LIN {X 0,Y 474.661,Z 275.668,A -85,B 0,C 180,E1 -7353.629,E2 -7353.629} C_VEL
LIN {X 0,Y 474.637,Z 275.665,A -85,B 0,C 180,E1 -7356.642,E2 -7356.642} C_VEL
LIN {X 0,Y 474.656,Z 275.67,A -85,B 0,C 180,E1 -7360.09,E2 -7360.09} C_VEL
LIN {X 0,Y 474.648,Z 275.66,A -85,B 0,C 180,E1 -7362.775,E2 -7362.775} C_VEL
LIN {X 0,Y 474.647,Z 275.67,A -85,B 0,C 180,E1 -7365.421,E2 -7365.421} C_VEL
LIN {X 0,Y 474.706,Z 275.661,A -85,B 0,C 180,E1 -7368.038,E2 -7368.038} C_VEL
LIN {X 0,Y 474.71,Z 275.661,A -85,B 0,C 180,E1 -7371.487,E2 -7371.487} C_VEL
LIN {X 0,Y 474.743,Z 275.645,A -85,B 0,C 180,E1 -7374.905,E2 -7374.905} C_VEL
LIN {X 0,Y 474.887,Z 275.637,A -85,B 0,C 180,E1 -7377.456,E2 -7377.456} C_VEL
LIN {X 0,Y 474.911,Z 275.639,A -85,B 0,C 180,E1 -7380,E2 -7380} C_VEL
LIN {X 0,Y 474.877,Z 275.632,A -85,B 0,C 180,E1 -7382.545,E2 -7382.545} C_VEL
LIN {X 0,Y 474.749,Z 275.66,A -85,B 0,C 180,E1 -7385.948,E2 -7385.948} C_VEL
LIN {X 0,Y 474.698,Z 275.655,A -85,B 0,C 180,E1 -7388.515,E2 -7388.515} C_VEL
LIN {X 0,Y 474.707,Z 275.667,A -85,B 0,C 180,E1 -7391.963,E2 -7391.963} C_VEL
LIN {X 0,Y 474.691,Z 275.662,A -85,B 0,C 180,E1 -7395.456,E2 -7395.456} C_VEL
LIN {X 0,Y 474.661,Z 275.656,A -85,B 0,C 180,E1 -7399.011,E2 -7399.011} C_VEL
LIN {X 0,Y 474.586,Z 275.681,A -85,B 0,C 180,E1 -7401.73,E2 -7401.73} C_VEL
LIN {X 0,Y 474.623,Z 275.67,A -85,B 0,C 180,E1 -7404.495,E2 -7404.495} C_VEL
LIN {X 0,Y 474.595,Z 275.676,A -85,B 0,C 180,E1 -7407.327,E2 -7407.327} C_VEL
LIN {X 0,Y 474.553,Z 275.688,A -85,B 0,C 180,E1 -7410.234,E2 -7410.234} C_VEL
LIN {X 0,Y 474.61,Z 275.676,A -85,B 0,C 180,E1 -7413.223,E2 -7413.223} C_VEL
LIN {X 0,Y 474.565,Z 275.685,A -85,B 0,C 180,E1 -7416.326,E2 -7416.326} C_VEL
LIN {X 0,Y 474.6,Z 275.68,A -85,B 0,C 180,E1 -7419.551,E2 -7419.551} C_VEL
LIN {X 0,Y 474.568,Z 275.682,A -85,B 0,C 180,E1 -7422.94,E2 -7422.94} C_VEL
LIN {X 0,Y 474.582,Z 275.68,A -85,B 0,C 180,E1 -7425.892,E2 -7425.892} C_VEL
LIN {X 0,Y 474.598,Z 275.757,A -85,B 0,C 180,E1 -7426.52,E2 -7426.52} C_VEL
LIN {X 0,Y 477.677,Z 285.882,A -85,B 0,C 180,E1 -7428.043,E2 -7428.043} C_VEL
LIN {X 0,Y 486.034,Z 303.231,A -85,B 0,C 180,E1 -7428.924,E2 -7428.924} C_VEL
LIN {X 0,Y 486.81,Z 305.51,A -85,B 0,C 180,E1 -7429.015,E2 -7429.015} C_VEL
LIN {X 0,Y 484.879,Z 443.516,A -85,B 0,C 180,E1 -7431.179,E2 -7431.179} C_VEL
LIN {X 0,Y 484.222,Z 449.369,A -85,B 0,C 180,E1 -7431.235,E2 -7431.235} C_VEL
LIN {X 0,Y 478.792,Z 468.46,A -85,B 0,C 180,E1 -7431.216,E2 -7431.216} C_VEL
LIN {X 0,Y 478.144,Z 474.313,A -85,B 0,C 180,E1 -7431.273,E2 -7431.273} C_VEL
LIN {X 0,Y 477.665,Z 496.241,A -85,B 0,C 180,E1 -7431.674,E2 -7431.674} C_VEL
LIN {X 0,Y 477.021,Z 512.96,A -85,B 0,C 180,E1 -7432.157,E2 -7432.157} C_VEL
LIN {X 0,Y 476.29,Z 528.431,A -85,B 0,C 180,E1 -7432.772,E2 -7432.772} C_VEL
LIN {X 0,Y 475.249,Z 544.663,A -85,B 0,C 180,E1 -7433.609,E2 -7433.609} C_VEL
LIN {X 0,Y 474.176,Z 559.577,A -85,B 0,C 180,E1 -7434.57,E2 -7434.57} C_VEL
LIN {X 0,Y 473.106,Z 573.275,A -85,B 0,C 180,E1 -7435.633,E2 -7435.633} C_VEL
LIN {X 0,Y 472.039,Z 586.323,A -85,B 0,C 180,E1 -7436.828,E2 -7436.828} C_VEL
LIN {X 0,Y 470.902,Z 599.014,A -85,B 0,C 180,E1 -7438.202,E2 -7438.202} C_VEL
LIN {X 0,Y 469.898,Z 610.493,A -85,B 0,C 180,E1 -7439.669,E2 -7439.669} C_VEL
LIN {X 0,Y 468.991,Z 621.639,A -85,B 0,C 180,E1 -7441.345,E2 -7441.345} C_VEL
LIN {X 0,Y 468.276,Z 630.97,A -85,B 0,C 180,E1 -7442.999,E2 -7442.999} C_VEL
LIN {X 0,Y 467.695,Z 639.197,A -85,B 0,C 180,E1 -7444.723,E2 -7444.723} C_VEL
LIN {X 0,Y 467.236,Z 646.457,A -85,B 0,C 180,E1 -7446.57,E2 -7446.57} C_VEL
LIN {X 0,Y 466.954,Z 652.215,A -85,B 0,C 180,E1 -7448.362,E2 -7448.362} C_VEL
LIN {X 0,Y 466.777,Z 656.937,A -85,B 0,C 180,E1 -7450.198,E2 -7450.198} C_VEL
LIN {X 0,Y 466.576,Z 661.108,A -85,B 0,C 180,E1 -7452.467,E2 -7452.467} C_VEL
LIN {X 0,Y 466.537,Z 663.472,A -85,B 0,C 180,E1 -7454.605,E2 -7454.605} C_VEL
LIN {X 0,Y 466.502,Z 664.25,A -85,B 0,C 180,E1 -7456.052,E2 -7456.052} C_VEL
LIN {X 0,Y 466.647,Z 664.195,A -85,B 0,C 180,E1 -7458.224,E2 -7458.224} C_VEL
LIN {X 0,Y 466.535,Z 662.564,A -85,B 0,C 180,E1 -7460.462,E2 -7460.462} C_VEL
LIN {X 0,Y 466.638,Z 660.118,A -85,B 0,C 180,E1 -7462.21,E2 -7462.21} C_VEL
LIN {X 0,Y 466.834,Z 656.756,A -85,B 0,C 180,E1 -7463.951,E2 -7463.951} C_VEL
LIN {X 0,Y 467.026,Z 651.048,A -85,B 0,C 180,E1 -7466.117,E2 -7466.117} C_VEL
LIN {X 0,Y 467.344,Z 643.603,A -85,B 0,C 180,E1 -7468.276,E2 -7468.276} C_VEL
LIN {X 0,Y 467.92,Z 635.211,A -85,B 0,C 180,E1 -7470.215,E2 -7470.215} C_VEL
LIN {X 0,Y 468.5,Z 626.235,A -85,B 0,C 180,E1 -7471.934,E2 -7471.934} C_VEL
LIN {X 0,Y 469.405,Z 615.604,A -85,B 0,C 180,E1 -7473.648,E2 -7473.648} C_VEL
LIN {X 0,Y 470.337,Z 604.684,A -85,B 0,C 180,E1 -7475.144,E2 -7475.144} C_VEL
LIN {X 0,Y 471.253,Z 593.821,A -85,B 0,C 180,E1 -7476.422,E2 -7476.422} C_VEL
LIN {X 0,Y 472.226,Z 581.157,A -85,B 0,C 180,E1 -7477.697,E2 -7477.697} C_VEL
LIN {X 0,Y 473.302,Z 567.479,A -85,B 0,C 180,E1 -7478.862,E2 -7478.862} C_VEL
LIN {X 0,Y 474.306,Z 554.277,A -85,B 0,C 180,E1 -7479.811,E2 -7479.811} C_VEL
LIN {X 0,Y 475.239,Z 540.053,A -85,B 0,C 180,E1 -7480.653,E2 -7480.653} C_VEL
LIN {X 0,Y 476.07,Z 524.768,A -85,B 0,C 180,E1 -7481.388,E2 -7481.388} C_VEL
LIN {X 0,Y 476.866,Z 508.398,A -85,B 0,C 180,E1 -7481.988,E2 -7481.988} C_VEL
LIN {X 0,Y 477.425,Z 492.53,A -85,B 0,C 180,E1 -7482.405,E2 -7482.405} C_VEL
LIN {X 0,Y 478.233,Z 435.094,A -85,B 0,C 180,E1 -7483.329,E2 -7483.329} C_VEL
LIN {X 0,Y 480.033,Z 307.307,A -85,B 0,C 180,E1 -7485.325,E2 -7485.325} C_VEL
LIN {X 0,Y 473.3,Z 292.179,A -85,B 0,C 180,E1 -7485.994,E2 -7485.994} C_VEL
LIN {X 0,Y 470.234,Z 285.606,A -85,B 0,C 180,E1 -7486.308,E2 -7486.308} C_VEL
LIN {X 0,Y 467.603,Z 276.551,A -85,B 0,C 180,E1 -7487.634,E2 -7487.634} C_VEL
LIN {X 0,Y 467.623,Z 276.551,A -85,B 0,C 180,E1 -7490.223,E2 -7490.223} C_VEL
LIN {X 0,Y 467.558,Z 276.562,A -85,B 0,C 180,E1 -7493.944,E2 -7493.944} C_VEL
LIN {X 0,Y 467.529,Z 276.559,A -85,B 0,C 180,E1 -7496.806,E2 -7496.806} C_VEL
LIN {X 0,Y 467.538,Z 276.559,A -85,B 0,C 180,E1 -7499.739,E2 -7499.739} C_VEL
LIN {X 0,Y 467.552,Z 276.556,A -85,B 0,C 180,E1 -7502.761,E2 -7502.761} C_VEL
LIN {X 0,Y 467.538,Z 276.558,A -85,B 0,C 180,E1 -7505.891,E2 -7505.891} C_VEL
LIN {X 0,Y 467.527,Z 276.555,A -85,B 0,C 180,E1 -7509.15,E2 -7509.15} C_VEL
LIN {X 0,Y 467.551,Z 276.554,A -85,B 0,C 180,E1 -7511.406,E2 -7511.406} C_VEL
LIN {X 0,Y 467.564,Z 276.552,A -85,B 0,C 180,E1 -7515.051,E2 -7515.051} C_VEL
LIN {X 0,Y 467.551,Z 276.554,A -85,B 0,C 180,E1 -7518.727,E2 -7518.727} C_VEL
LIN {X 0,Y 467.54,Z 276.54,A -85,B 0,C 180,E1 -7521.952,E2 -7521.952} C_VEL
LIN {X 0,Y 467.551,Z 276.54,A -85,B 0,C 180,E1 -7525.166,E2 -7525.166} C_VEL
LIN {X 0,Y 467.559,Z 276.555,A -85,B 0,C 180,E1 -7528.257,E2 -7528.257} C_VEL
LIN {X 0,Y 467.544,Z 276.548,A -85,B 0,C 180,E1 -7531.248,E2 -7531.248} C_VEL
LIN {X 0,Y 467.577,Z 276.549,A -85,B 0,C 180,E1 -7534.401,E2 -7534.401} C_VEL
LIN {X 0,Y 467.577,Z 276.544,A -85,B 0,C 180,E1 -7536.995,E2 -7536.995} C_VEL
LIN {X 0,Y 467.623,Z 276.549,A -85,B 0,C 180,E1 -7539.777,E2 -7539.777} C_VEL
LIN {X 0,Y 467.595,Z 276.541,A -85,B 0,C 180,E1 -7542.506,E2 -7542.506} C_VEL
LIN {X 0,Y 467.602,Z 276.55,A -85,B 0,C 180,E1 -7545.196,E2 -7545.196} C_VEL
LIN {X 0,Y 467.658,Z 276.536,A -85,B 0,C 180,E1 -7547.854,E2 -7547.854} C_VEL
LIN {X 0,Y 467.669,Z 276.544,A -85,B 0,C 180,E1 -7551.357,E2 -7551.357} C_VEL
LIN {X 0,Y 467.736,Z 276.524,A -85,B 0,C 180,E1 -7553.962,E2 -7553.962} C_VEL
LIN {X 0,Y 467.849,Z 276.524,A -85,B 0,C 180,E1 -7557.417,E2 -7557.417} C_VEL
LIN {X 0,Y 467.882,Z 276.504,A -85,B 0,C 180,E1 -7560,E2 -7560} C_VEL
LIN {X 0,Y 467.859,Z 276.514,A -85,B 0,C 180,E1 -7562.582,E2 -7562.582} C_VEL
LIN {X 0,Y 467.724,Z 276.523,A -85,B 0,C 180,E1 -7566.037,E2 -7566.037} C_VEL
LIN {X 0,Y 467.682,Z 276.532,A -85,B 0,C 180,E1 -7568.642,E2 -7568.642} C_VEL
LIN {X 0,Y 467.656,Z 276.538,A -85,B 0,C 180,E1 -7572.145,E2 -7572.145} C_VEL
LIN {X 0,Y 467.639,Z 276.544,A -85,B 0,C 180,E1 -7575.695,E2 -7575.695} C_VEL
LIN {X 0,Y 467.622,Z 276.55,A -85,B 0,C 180,E1 -7579.307,E2 -7579.307} C_VEL
LIN {X 0,Y 467.534,Z 276.555,A -85,B 0,C 180,E1 -7582.073,E2 -7582.073} C_VEL
LIN {X 0,Y 467.604,Z 276.554,A -85,B 0,C 180,E1 -7584.887,E2 -7584.887} C_VEL
LIN {X 0,Y 467.619,Z 276.544,A -85,B 0,C 180,E1 -7587.769,E2 -7587.769} C_VEL
LIN {X 0,Y 467.567,Z 276.557,A -85,B 0,C 180,E1 -7591.045,E2 -7591.045} C_VEL
LIN {X 0,Y 467.588,Z 276.55,A -85,B 0,C 180,E1 -7594.242,E2 -7594.242} C_VEL
LIN {X 0,Y 467.549,Z 276.554,A -85,B 0,C 180,E1 -7597.186,E2 -7597.186} C_VEL
LIN {X 0,Y 467.577,Z 276.55,A -85,B 0,C 180,E1 -7600.264,E2 -7600.264} C_VEL
LIN {X 0,Y 467.585,Z 276.554,A -85,B 0,C 180,E1 -7602.567,E2 -7602.567} C_VEL
LIN {X 0,Y 467.569,Z 276.555,A -85,B 0,C 180,E1 -7605.053,E2 -7605.053} C_VEL
LIN {X 0,Y 467.587,Z 276.549,A -85,B 0,C 180,E1 -7607.44,E2 -7607.44} C_VEL
LIN {X 0,Y 467.581,Z 276.556,A -85,B 0,C 180,E1 -7610.855,E2 -7610.855} C_VEL
LIN {X 0,Y 467.558,Z 276.554,A -85,B 0,C 180,E1 -7614.261,E2 -7614.261} C_VEL
LIN {X 0,Y 467.62,Z 276.653,A -85,B 0,C 180,E1 -7616.939,E2 -7616.939} C_VEL
LIN {X 0,Y 474.089,Z 297.974,A -85,B 0,C 180,E1 -7619.734,E2 -7619.734} C_VEL
LIN {X 0,Y 475.758,Z 304.134,A -85,B 0,C 180,E1 -7620.503,E2 -7620.503} C_VEL
LIN {X 0,Y 475.416,Z 309.361,A -85,B 0,C 180,E1 -7621.045,E2 -7621.045} C_VEL
LIN {X 0,Y 479.849,Z 335.021,A -85,B 0,C 180,E1 -7621.748,E2 -7621.748} C_VEL
LIN {X 0,Y 477.322,Z 515.075,A -85,B 0,C 180,E1 -7624.569,E2 -7624.569} C_VEL
LIN {X 0,Y 476.755,Z 530.976,A -85,B 0,C 180,E1 -7624.954,E2 -7624.954} C_VEL
LIN {X 0,Y 476.072,Z 547.463,A -85,B 0,C 180,E1 -7625.527,E2 -7625.527} C_VEL
LIN {X 0,Y 475.182,Z 561.942,A -85,B 0,C 180,E1 -7626.174,E2 -7626.174} C_VEL
LIN {X 0,Y 474.26,Z 575.705,A -85,B 0,C 180,E1 -7626.948,E2 -7626.948} C_VEL
LIN {X 0,Y 473.097,Z 590.803,A -85,B 0,C 180,E1 -7627.97,E2 -7627.97} C_VEL
LIN {X 0,Y 472.056,Z 604.285,A -85,B 0,C 180,E1 -7629.065,E2 -7629.065} C_VEL
LIN {X 0,Y 470.947,Z 618.3,A -85,B 0,C 180,E1 -7630.426,E2 -7630.426} C_VEL
LIN {X 0,Y 470.025,Z 629.422,A -85,B 0,C 180,E1 -7631.7,E2 -7631.7} C_VEL
LIN {X 0,Y 469.126,Z 640.999,A -85,B 0,C 180,E1 -7633.239,E2 -7633.239} C_VEL
LIN {X 0,Y 468.442,Z 650.925,A -85,B 0,C 180,E1 -7634.779,E2 -7634.779} C_VEL
LIN {X 0,Y 467.748,Z 660.458,A -85,B 0,C 180,E1 -7636.533,E2 -7636.533} C_VEL
LIN {X 0,Y 467.359,Z 668.439,A -85,B 0,C 180,E1 -7638.287,E2 -7638.287} C_VEL
LIN {X 0,Y 466.981,Z 675.094,A -85,B 0,C 180,E1 -7640.034,E2 -7640.034} C_VEL
LIN {X 0,Y 466.833,Z 680.492,A -85,B 0,C 180,E1 -7641.778,E2 -7641.778} C_VEL
LIN {X 0,Y 466.748,Z 684.944,A -85,B 0,C 180,E1 -7643.607,E2 -7643.607} C_VEL
LIN {X 0,Y 466.605,Z 688.611,A -85,B 0,C 180,E1 -7645.681,E2 -7645.681} C_VEL
LIN {X 0,Y 466.637,Z 690.554,A -85,B 0,C 180,E1 -7647.41,E2 -7647.41} C_VEL
LIN {X 0,Y 466.614,Z 691.515,A -85,B 0,C 180,E1 -7649.137,E2 -7649.137} C_VEL
LIN {X 0,Y 466.615,Z 691.51,A -85,B 0,C 180,E1 -7650.863,E2 -7650.863} C_VEL
LIN {X 0,Y 466.637,Z 690.539,A -85,B 0,C 180,E1 -7652.59,E2 -7652.59} C_VEL
LIN {X 0,Y 466.606,Z 688.587,A -85,B 0,C 180,E1 -7654.319,E2 -7654.319} C_VEL
LIN {X 0,Y 466.748,Z 684.913,A -85,B 0,C 180,E1 -7656.394,E2 -7656.394} C_VEL
LIN {X 0,Y 466.794,Z 680.451,A -85,B 0,C 180,E1 -7658.223,E2 -7658.223} C_VEL
LIN {X 0,Y 466.981,Z 675.045,A -85,B 0,C 180,E1 -7659.967,E2 -7659.967} C_VEL
LIN {X 0,Y 467.359,Z 668.384,A -85,B 0,C 180,E1 -7661.713,E2 -7661.713} C_VEL
LIN {X 0,Y 467.741,Z 660.409,A -85,B 0,C 180,E1 -7663.468,E2 -7663.468} C_VEL
LIN {X 0,Y 468.436,Z 650.897,A -85,B 0,C 180,E1 -7665.222,E2 -7665.222} C_VEL
LIN {X 0,Y 469.265,Z 639.518,A -85,B 0,C 180,E1 -7666.98,E2 -7666.98} C_VEL
LIN {X 0,Y 470.235,Z 627.72,A -85,B 0,C 180,E1 -7668.518,E2 -7668.518} C_VEL
LIN {X 0,Y 471.238,Z 615.457,A -85,B 0,C 180,E1 -7669.884,E2 -7669.884} C_VEL
LIN {X 0,Y 472.335,Z 602.13,A -85,B 0,C 180,E1 -7671.151,E2 -7671.151} C_VEL
LIN {X 0,Y 473.386,Z 588.501,A -85,B 0,C 180,E1 -7672.246,E2 -7672.246} C_VEL
LIN {X 0,Y 474.485,Z 574.417,A -85,B 0,C 180,E1 -7673.183,E2 -7673.183} C_VEL
LIN {X 0,Y 475.561,Z 558.809,A -85,B 0,C 180,E1 -7674.037,E2 -7674.037} C_VEL
LIN {X 0,Y 476.477,Z 543.201,A -85,B 0,C 180,E1 -7674.713,E2 -7674.713} C_VEL
LIN {X 0,Y 477.276,Z 526.491,A -85,B 0,C 180,E1 -7675.25,E2 -7675.25} C_VEL
LIN {X 0,Y 477.79,Z 509.954,A -85,B 0,C 180,E1 -7675.603,E2 -7675.603} C_VEL
LIN {X 0,Y 480.42,Z 335.028,A -85,B 0,C 180,E1 -7678.373,E2 -7678.373} C_VEL
LIN {X 0,Y 476.597,Z 313.02,A -85,B 0,C 180,E1 -7679.018,E2 -7679.018} C_VEL
LIN {X 0,Y 475.858,Z 308.841,A -85,B 0,C 180,E1 -7679.169,E2 -7679.169} C_VEL
LIN {X 0,Y 476.125,Z 304.227,A -85,B 0,C 180,E1 -7679.665,E2 -7679.665} C_VEL
LIN {X 0,Y 471.964,Z 289.925,A -85,B 0,C 180,E1 -7681.599,E2 -7681.599} C_VEL
LIN {X 0,Y 467.609,Z 276.551,A -85,B 0,C 180,E1 -7683.56,E2 -7683.56} C_VEL
LIN {X 0,Y 467.528,Z 276.557,A -85,B 0,C 180,E1 -7686.962,E2 -7686.962} C_VEL
LIN {X 0,Y 467.582,Z 276.553,A -85,B 0,C 180,E1 -7689.955,E2 -7689.955} C_VEL
LIN {X 0,Y 467.586,Z 276.546,A -85,B 0,C 180,E1 -7692.567,E2 -7692.567} C_VEL
LIN {X 0,Y 467.57,Z 276.549,A -85,B 0,C 180,E1 -7695.054,E2 -7695.054} C_VEL
LIN {X 0,Y 467.588,Z 276.549,A -85,B 0,C 180,E1 -7697.44,E2 -7697.44} C_VEL
LIN {X 0,Y 467.582,Z 276.557,A -85,B 0,C 180,E1 -7700.856,E2 -7700.856} C_VEL
LIN {X 0,Y 467.559,Z 276.553,A -85,B 0,C 180,E1 -7704.261,E2 -7704.261} C_VEL
LIN {X 0,Y 467.582,Z 276.545,A -85,B 0,C 180,E1 -7707.321,E2 -7707.321} C_VEL
LIN {X 0,Y 467.57,Z 276.55,A -85,B 0,C 180,E1 -7710.668,E2 -7710.668} C_VEL
LIN {X 0,Y 467.618,Z 276.546,A -85,B 0,C 180,E1 -7713.2,E2 -7713.2} C_VEL
LIN {X 0,Y 467.594,Z 276.544,A -85,B 0,C 180,E1 -7716.469,E2 -7716.469} C_VEL
LIN {X 0,Y 467.624,Z 276.545,A -85,B 0,C 180,E1 -7719.778,E2 -7719.778} C_VEL
LIN {X 0,Y 467.607,Z 276.539,A -85,B 0,C 180,E1 -7722.507,E2 -7722.507} C_VEL
LIN {X 0,Y 467.606,Z 276.549,A -85,B 0,C 180,E1 -7725.197,E2 -7725.197} C_VEL
LIN {X 0,Y 467.658,Z 276.538,A -85,B 0,C 180,E1 -7727.855,E2 -7727.855} C_VEL
LIN {X 0,Y 467.669,Z 276.539,A -85,B 0,C 180,E1 -7731.357,E2 -7731.357} C_VEL
LIN {X 0,Y 467.715,Z 276.533,A -85,B 0,C 180,E1 -7733.963,E2 -7733.963} C_VEL
LIN {X 0,Y 467.852,Z 276.513,A -85,B 0,C 180,E1 -7737.418,E2 -7737.418} C_VEL
LIN {X 0,Y 467.88,Z 276.515,A -85,B 0,C 180,E1 -7740,E2 -7740} C_VEL
LIN {X 0,Y 467.817,Z 276.511,A -85,B 0,C 180,E1 -7742.584,E2 -7742.584} C_VEL
LIN {X 0,Y 467.712,Z 276.538,A -85,B 0,C 180,E1 -7746.038,E2 -7746.038} C_VEL
LIN {X 0,Y 467.659,Z 276.532,A -85,B 0,C 180,E1 -7748.644,E2 -7748.644} C_VEL
LIN {X 0,Y 467.659,Z 276.542,A -85,B 0,C 180,E1 -7752.146,E2 -7752.146} C_VEL
LIN {X 0,Y 467.616,Z 276.545,A -85,B 0,C 180,E1 -7755.696,E2 -7755.696} C_VEL
LIN {X 0,Y 467.621,Z 276.532,A -85,B 0,C 180,E1 -7759.308,E2 -7759.308} C_VEL
LIN {X 0,Y 467.529,Z 276.562,A -85,B 0,C 180,E1 -7762.075,E2 -7762.075} C_VEL
LIN {X 0,Y 467.553,Z 276.552,A -85,B 0,C 180,E1 -7764.891,E2 -7764.891} C_VEL
LIN {X 0,Y 467.54,Z 276.553,A -85,B 0,C 180,E1 -7767.775,E2 -7767.775} C_VEL
LIN {X 0,Y 467.53,Z 276.557,A -85,B 0,C 180,E1 -7771.037,E2 -7771.037} C_VEL
LIN {X 0,Y 467.564,Z 276.557,A -85,B 0,C 180,E1 -7774.237,E2 -7774.237} C_VEL
LIN {X 0,Y 467.511,Z 276.564,A -85,B 0,C 180,E1 -7777.18,E2 -7777.18} C_VEL
LIN {X 0,Y 467.52,Z 276.561,A -85,B 0,C 180,E1 -7780.271,E2 -7780.271} C_VEL
LIN {X 0,Y 467.519,Z 276.561,A -85,B 0,C 180,E1 -7782.569,E2 -7782.569} C_VEL
LIN {X 0,Y 467.557,Z 276.554,A -85,B 0,C 180,E1 -7785.878,E2 -7785.878} C_VEL
LIN {X 0,Y 467.571,Z 276.74,A -85,B 0,C 180,E1 -7786.065,E2 -7786.065} C_VEL
LIN {X 0,Y 470.647,Z 286.352,A -85,B 0,C 180,E1 -7787.53,E2 -7787.53} C_VEL
LIN {X 0,Y 479.664,Z 304.887,A -85,B 0,C 180,E1 -7788.511,E2 -7788.511} C_VEL
LIN {X 0,Y 480.616,Z 306.974,A -85,B 0,C 180,E1 -7788.614,E2 -7788.614} C_VEL
LIN {X 0,Y 479.557,Z 380.616,A -85,B 0,C 180,E1 -7789.793,E2 -7789.793} C_VEL
LIN {X 0,Y 478.144,Z 474.313,A -85,B 0,C 180,E1 -7791.273,E2 -7791.273} C_VEL
LIN {X 0,Y 477.526,Z 480.156,A -85,B 0,C 180,E1 -7791.331,E2 -7791.331} C_VEL
LIN {X 0,Y 472.521,Z 497.266,A -85,B 0,C 180,E1 -7791.378,E2 -7791.378} C_VEL
LIN {X 0,Y 471.265,Z 503.014,A -85,B 0,C 180,E1 -7791.462,E2 -7791.462} C_VEL
LIN {X 0,Y 471.06,Z 504.923,A -85,B 0,C 180,E1 -7791.512,E2 -7791.512} C_VEL
LIN {X 0,Y 470.373,Z 519.803,A -85,B 0,C 180,E1 -7792.019,E2 -7792.019} C_VEL
LIN {X 0,Y 469.458,Z 534.84,A -85,B 0,C 180,E1 -7792.7,E2 -7792.7} C_VEL
LIN {X 0,Y 468.47,Z 549.447,A -85,B 0,C 180,E1 -7793.526,E2 -7793.526} C_VEL
LIN {X 0,Y 467.331,Z 564.147,A -85,B 0,C 180,E1 -7794.539,E2 -7794.539} C_VEL
LIN {X 0,Y 466.144,Z 578.17,A -85,B 0,C 180,E1 -7795.702,E2 -7795.702} C_VEL
LIN {X 0,Y 464.881,Z 591.514,A -85,B 0,C 180,E1 -7797.027,E2 -7797.027} C_VEL
LIN {X 0,Y 463.723,Z 603.844,A -85,B 0,C 180,E1 -7798.475,E2 -7798.475} C_VEL
LIN {X 0,Y 462.667,Z 615.421,A -85,B 0,C 180,E1 -7800.075,E2 -7800.075} C_VEL
LIN {X 0,Y 461.861,Z 624.919,A -85,B 0,C 180,E1 -7801.607,E2 -7801.607} C_VEL
LIN {X 0,Y 461.041,Z 634.892,A -85,B 0,C 180,E1 -7803.52,E2 -7803.52} C_VEL
LIN {X 0,Y 460.508,Z 642.099,A -85,B 0,C 180,E1 -7805.185,E2 -7805.185} C_VEL
LIN {X 0,Y 460.099,Z 648.942,A -85,B 0,C 180,E1 -7807.076,E2 -7807.076} C_VEL
LIN {X 0,Y 459.847,Z 654.016,A -85,B 0,C 180,E1 -7808.795,E2 -7808.795} C_VEL
LIN {X 0,Y 459.669,Z 657.665,A -85,B 0,C 180,E1 -7810.344,E2 -7810.344} C_VEL
LIN {X 0,Y 459.506,Z 660.994,A -85,B 0,C 180,E1 -7812.188,E2 -7812.188} C_VEL
LIN {X 0,Y 459.461,Z 663.629,A -85,B 0,C 180,E1 -7814.508,E2 -7814.508} C_VEL
LIN {X 0,Y 459.422,Z 664.407,A -85,B 0,C 180,E1 -7815.832,E2 -7815.832} C_VEL
LIN {X 0,Y 459.561,Z 664.425,A -85,B 0,C 180,E1 -7818.168,E2 -7818.168} C_VEL
LIN {X 0,Y 459.507,Z 663.749,A -85,B 0,C 180,E1 -7819.424,E2 -7819.424} C_VEL
LIN {X 0,Y 459.484,Z 661.911,A -85,B 0,C 180,E1 -7821.202,E2 -7821.202} C_VEL
LIN {X 0,Y 459.616,Z 659.157,A -85,B 0,C 180,E1 -7822.973,E2 -7822.973} C_VEL
LIN {X 0,Y 459.767,Z 655.324,A -85,B 0,C 180,E1 -7824.738,E2 -7824.738} C_VEL
LIN {X 0,Y 460.015,Z 650.476,A -85,B 0,C 180,E1 -7826.496,E2 -7826.496} C_VEL
LIN {X 0,Y 460.266,Z 644.512,A -85,B 0,C 180,E1 -7828.25,E2 -7828.25} C_VEL
LIN {X 0,Y 460.779,Z 637.26,A -85,B 0,C 180,E1 -7830,E2 -7830} C_VEL
LIN {X 0,Y 461.35,Z 628.68,A -85,B 0,C 180,E1 -7831.746,E2 -7831.746} C_VEL
LIN {X 0,Y 462.275,Z 618.49,A -85,B 0,C 180,E1 -7833.486,E2 -7833.486} C_VEL
LIN {X 0,Y 463.241,Z 607.946,A -85,B 0,C 180,E1 -7835.004,E2 -7835.004} C_VEL
LIN {X 0,Y 464.328,Z 595.614,A -85,B 0,C 180,E1 -7836.518,E2 -7836.518} C_VEL
LIN {X 0,Y 465.364,Z 583.247,A -85,B 0,C 180,E1 -7837.812,E2 -7837.812} C_VEL
LIN {X 0,Y 466.489,Z 569.949,A -85,B 0,C 180,E1 -7838.993,E2 -7838.993} C_VEL
LIN {X 0,Y 467.612,Z 555.453,A -85,B 0,C 180,E1 -7840.062,E2 -7840.062} C_VEL
LIN {X 0,Y 468.575,Z 541.449,A -85,B 0,C 180,E1 -7840.915,E2 -7840.915} C_VEL
LIN {X 0,Y 469.44,Z 526.508,A -85,B 0,C 180,E1 -7841.66,E2 -7841.66} C_VEL
LIN {X 0,Y 470.323,Z 509.858,A -85,B 0,C 180,E1 -7842.294,E2 -7842.294} C_VEL
LIN {X 0,Y 470.937,Z 494.262,A -85,B 0,C 180,E1 -7842.716,E2 -7842.716} C_VEL
LIN {X 0,Y 471.372,Z 469.837,A -85,B 0,C 180,E1 -7843.142,E2 -7843.142} C_VEL
LIN {X 0,Y 473.675,Z 310.27,A -85,B 0,C 180,E1 -7845.666,E2 -7845.666} C_VEL
LIN {X 0,Y 473.394,Z 308.272,A -85,B 0,C 180,E1 -7845.717,E2 -7845.717} C_VEL
LIN {X 0,Y 463.002,Z 285.891,A -85,B 0,C 180,E1 -7846.762,E2 -7846.762} C_VEL
LIN {X 0,Y 460.574,Z 277.428,A -85,B 0,C 180,E1 -7848.028,E2 -7848.028} C_VEL
LIN {X 0,Y 460.553,Z 277.432,A -85,B 0,C 180,E1 -7850.547,E2 -7850.547} C_VEL
LIN {X 0,Y 460.531,Z 277.435,A -85,B 0,C 180,E1 -7853.702,E2 -7853.702} C_VEL
LIN {X 0,Y 460.482,Z 277.431,A -85,B 0,C 180,E1 -7856.27,E2 -7856.27} C_VEL
LIN {X 0,Y 460.519,Z 277.432,A -85,B 0,C 180,E1 -7859.232,E2 -7859.232} C_VEL
LIN {X 0,Y 460.503,Z 277.436,A -85,B 0,C 180,E1 -7862.287,E2 -7862.287} C_VEL
LIN {X 0,Y 460.494,Z 277.43,A -85,B 0,C 180,E1 -7865.447,E2 -7865.447} C_VEL
LIN {X 0,Y 460.48,Z 277.433,A -85,B 0,C 180,E1 -7868.887,E2 -7868.887} C_VEL
LIN {X 0,Y 460.497,Z 277.435,A -85,B 0,C 180,E1 -7871.597,E2 -7871.597} C_VEL
LIN {X 0,Y 460.508,Z 277.432,A -85,B 0,C 180,E1 -7874.59,E2 -7874.59} C_VEL
LIN {X 0,Y 460.472,Z 277.437,A -85,B 0,C 180,E1 -7877.812,E2 -7877.812} C_VEL
LIN {X 0,Y 460.496,Z 277.432,A -85,B 0,C 180,E1 -7880.133,E2 -7880.133} C_VEL
LIN {X 0,Y 460.46,Z 277.413,A -85,B 0,C 180,E1 -7883.468,E2 -7883.468} C_VEL
LIN {X 0,Y 460.518,Z 277.427,A -85,B 0,C 180,E1 -7886.674,E2 -7886.674} C_VEL
LIN {X 0,Y 460.504,Z 277.432,A -85,B 0,C 180,E1 -7889.759,E2 -7889.759} C_VEL
LIN {X 0,Y 460.49,Z 277.432,A -85,B 0,C 180,E1 -7892.75,E2 -7892.75} C_VEL
LIN {X 0,Y 460.518,Z 277.428,A -85,B 0,C 180,E1 -7895.666,E2 -7895.666} C_VEL
LIN {X 0,Y 460.523,Z 277.429,A -85,B 0,C 180,E1 -7898.578,E2 -7898.578} C_VEL
LIN {X 0,Y 460.587,Z 277.422,A -85,B 0,C 180,E1 -7901.31,E2 -7901.31} C_VEL
LIN {X 0,Y 460.606,Z 277.421,A -85,B 0,C 180,E1 -7904.059,E2 -7904.059} C_VEL
LIN {X 0,Y 460.611,Z 277.415,A -85,B 0,C 180,E1 -7907.665,E2 -7907.665} C_VEL
LIN {X 0,Y 460.619,Z 277.421,A -85,B 0,C 180,E1 -7911.223,E2 -7911.223} C_VEL
LIN {X 0,Y 460.702,Z 277.4,A -85,B 0,C 180,E1 -7913.869,E2 -7913.869} C_VEL
LIN {X 0,Y 460.789,Z 277.402,A -85,B 0,C 180,E1 -7917.377,E2 -7917.377} C_VEL
LIN {X 0,Y 460.852,Z 277.379,A -85,B 0,C 180,E1 -7920,E2 -7920} C_VEL
LIN {X 0,Y 460.8,Z 277.394,A -85,B 0,C 180,E1 -7922.622,E2 -7922.622} C_VEL
LIN {X 0,Y 460.688,Z 277.399,A -85,B 0,C 180,E1 -7926.13,E2 -7926.13} C_VEL
LIN {X 0,Y 460.629,Z 277.411,A -85,B 0,C 180,E1 -7928.776,E2 -7928.776} C_VEL
LIN {X 0,Y 460.614,Z 277.415,A -85,B 0,C 180,E1 -7932.444,E2 -7932.444} C_VEL
LIN {X 0,Y 460.6,Z 277.419,A -85,B 0,C 180,E1 -7935.997,E2 -7935.997} C_VEL
LIN {X 0,Y 460.568,Z 277.427,A -85,B 0,C 180,E1 -7939.615,E2 -7939.615} C_VEL
LIN {X 0,Y 460.511,Z 277.43,A -85,B 0,C 180,E1 -7942.428,E2 -7942.428} C_VEL
LIN {X 0,Y 460.567,Z 277.426,A -85,B 0,C 180,E1 -7945.802,E2 -7945.802} C_VEL
LIN {X 0,Y 460.552,Z 277.424,A -85,B 0,C 180,E1 -7948.233,E2 -7948.233} C_VEL
LIN {X 0,Y 460.52,Z 277.436,A -85,B 0,C 180,E1 -7951.283,E2 -7951.283} C_VEL
LIN {X 0,Y 460.532,Z 277.431,A -85,B 0,C 180,E1 -7954.506,E2 -7954.506} C_VEL
LIN {X 0,Y 460.527,Z 277.429,A -85,B 0,C 180,E1 -7957.62,E2 -7957.62} C_VEL
LIN {X 0,Y 460.541,Z 277.427,A -85,B 0,C 180,E1 -7960.269,E2 -7960.269} C_VEL
LIN {X 0,Y 460.509,Z 277.432,A -85,B 0,C 180,E1 -7963.374,E2 -7963.374} C_VEL
LIN {X 0,Y 460.508,Z 277.437,A -85,B 0,C 180,E1 -7966.626,E2 -7966.626} C_VEL
LIN {X 0,Y 460.541,Z 277.429,A -85,B 0,C 180,E1 -7969.73,E2 -7969.73} C_VEL
LIN {X 0,Y 460.498,Z 277.437,A -85,B 0,C 180,E1 -7972.524,E2 -7972.524} C_VEL
LIN {X 0,Y 460.544,Z 277.429,A -85,B 0,C 180,E1 -7975.624,E2 -7975.624} C_VEL
LIN {X 0,Y 460.609,Z 277.601,A -85,B 0,C 180,E1 -7976.551,E2 -7976.551} C_VEL
LIN {X 0,Y 466.856,Z 298.094,A -85,B 0,C 180,E1 -7979.289,E2 -7979.289} C_VEL
LIN {X 0,Y 469.068,Z 306.394,A -85,B 0,C 180,E1 -7980.343,E2 -7980.343} C_VEL
LIN {X 0,Y 468.902,Z 309.11,A -85,B 0,C 180,E1 -7980.63,E2 -7980.63} C_VEL
LIN {X 0,Y 473.5,Z 336.299,A -85,B 0,C 180,E1 -7981.385,E2 -7981.385} C_VEL
LIN {X 0,Y 470.826,Z 515.277,A -85,B 0,C 180,E1 -7984.225,E2 -7984.225} C_VEL
LIN {X 0,Y 470.194,Z 531.868,A -85,B 0,C 180,E1 -7984.639,E2 -7984.639} C_VEL
LIN {X 0,Y 469.514,Z 546.746,A -85,B 0,C 180,E1 -7985.162,E2 -7985.162} C_VEL
LIN {X 0,Y 468.543,Z 562.438,A -85,B 0,C 180,E1 -7985.874,E2 -7985.874} C_VEL
LIN {X 0,Y 467.506,Z 577.396,A -85,B 0,C 180,E1 -7986.74,E2 -7986.74} C_VEL
LIN {X 0,Y 466.323,Z 591.811,A -85,B 0,C 180,E1 -7987.749,E2 -7987.749} C_VEL
LIN {X 0,Y 465.127,Z 606.275,A -85,B 0,C 180,E1 -7988.97,E2 -7988.97} C_VEL
LIN {X 0,Y 464.117,Z 618.362,A -85,B 0,C 180,E1 -7990.17,E2 -7990.17} C_VEL
LIN {X 0,Y 463.005,Z 630.907,A -85,B 0,C 180,E1 -7991.641,E2 -7991.641} C_VEL
LIN {X 0,Y 462.09,Z 642.215,A -85,B 0,C 180,E1 -7993.204,E2 -7993.204} C_VEL
LIN {X 0,Y 461.366,Z 651.914,A -85,B 0,C 180,E1 -7994.766,E2 -7994.766} C_VEL
LIN {X 0,Y 460.693,Z 661.327,A -85,B 0,C 180,E1 -7996.547,E2 -7996.547} C_VEL
LIN {X 0,Y 460.186,Z 670.035,A -85,B 0,C 180,E1 -7998.549,E2 -7998.549} C_VEL
LIN {X 0,Y 459.786,Z 677.75,A -85,B 0,C 180,E1 -8000.764,E2 -8000.764} C_VEL
LIN {X 0,Y 459.648,Z 683.614,A -85,B 0,C 180,E1 -8002.974,E2 -8002.974} C_VEL
LIN {X 0,Y 459.577,Z 687.043,A -85,B 0,C 180,E1 -8004.736,E2 -8004.736} C_VEL
LIN {X 0,Y 459.56,Z 689.533,A -85,B 0,C 180,E1 -8006.493,E2 -8006.493} C_VEL
LIN {X 0,Y 459.511,Z 690.934,A -85,B 0,C 180,E1 -8008.247,E2 -8008.247} C_VEL
LIN {X 0,Y 459.525,Z 691.46,A -85,B 0,C 180,E1 -8010,E2 -8010} C_VEL
LIN {X 0,Y 459.533,Z 690.925,A -85,B 0,C 180,E1 -8011.753,E2 -8011.753} C_VEL
LIN {X 0,Y 459.56,Z 689.513,A -85,B 0,C 180,E1 -8013.507,E2 -8013.507} C_VEL
LIN {X 0,Y 459.577,Z 687.016,A -85,B 0,C 180,E1 -8015.265,E2 -8015.265} C_VEL
LIN {X 0,Y 459.648,Z 683.585,A -85,B 0,C 180,E1 -8017.026,E2 -8017.026} C_VEL
LIN {X 0,Y 459.786,Z 677.72,A -85,B 0,C 180,E1 -8019.236,E2 -8019.236} C_VEL
LIN {X 0,Y 460.186,Z 670.017,A -85,B 0,C 180,E1 -8021.452,E2 -8021.452} C_VEL
LIN {X 0,Y 460.651,Z 661.334,A -85,B 0,C 180,E1 -8023.454,E2 -8023.454} C_VEL
LIN {X 0,Y 461.361,Z 651.977,A -85,B 0,C 180,E1 -8025.235,E2 -8025.235} C_VEL
LIN {X 0,Y 462.1,Z 642.366,A -85,B 0,C 180,E1 -8026.796,E2 -8026.796} C_VEL
LIN {X 0,Y 463.056,Z 631.189,A -85,B 0,C 180,E1 -8028.357,E2 -8028.357} C_VEL
LIN {X 0,Y 464.186,Z 618.799,A -85,B 0,C 180,E1 -8029.827,E2 -8029.827} C_VEL
LIN {X 0,Y 465.285,Z 605.77,A -85,B 0,C 180,E1 -8031.139,E2 -8031.139} C_VEL
LIN {X 0,Y 466.532,Z 591.395,A -85,B 0,C 180,E1 -8032.357,E2 -8032.357} C_VEL
LIN {X 0,Y 467.771,Z 576.926,A -85,B 0,C 180,E1 -8033.376,E2 -8033.376} C_VEL
LIN {X 0,Y 468.925,Z 561.254,A -85,B 0,C 180,E1 -8034.282,E2 -8034.282} C_VEL
LIN {X 0,Y 469.931,Z 545.621,A -85,B 0,C 180,E1 -8034.992,E2 -8034.992} C_VEL
LIN {X 0,Y 470.74,Z 529.703,A -85,B 0,C 180,E1 -8035.537,E2 -8035.537} C_VEL
LIN {X 0,Y 471.386,Z 512.47,A -85,B 0,C 180,E1 -8035.945,E2 -8035.945} C_VEL
LIN {X 0,Y 474.263,Z 336.161,A -85,B 0,C 180,E1 -8038.783,E2 -8038.783} C_VEL
LIN {X 0,Y 469.939,Z 311.46,A -85,B 0,C 180,E1 -8039.53,E2 -8039.53} C_VEL
LIN {X 0,Y 469.525,Z 308.646,A -85,B 0,C 180,E1 -8039.635,E2 -8039.635} C_VEL
LIN {X 0,Y 469.457,Z 306.018,A -85,B 0,C 180,E1 -8039.938,E2 -8039.938} C_VEL
LIN {X 0,Y 465.265,Z 291.711,A -85,B 0,C 180,E1 -8041.917,E2 -8041.917} C_VEL
LIN {X 0,Y 460.558,Z 277.43,A -85,B 0,C 180,E1 -8044.045,E2 -8044.045} C_VEL
LIN {X 0,Y 460.526,Z 277.435,A -85,B 0,C 180,E1 -8047.621,E2 -8047.621} C_VEL
LIN {X 0,Y 460.542,Z 277.43,A -85,B 0,C 180,E1 -8050.27,E2 -8050.27} C_VEL
LIN {X 0,Y 460.509,Z 277.437,A -85,B 0,C 180,E1 -8053.375,E2 -8053.375} C_VEL
LIN {X 0,Y 460.5,Z 277.435,A -85,B 0,C 180,E1 -8056.625,E2 -8056.625} C_VEL
LIN {X 0,Y 460.542,Z 277.428,A -85,B 0,C 180,E1 -8059.731,E2 -8059.731} C_VEL
LIN {X 0,Y 460.499,Z 277.426,A -85,B 0,C 180,E1 -8062.524,E2 -8062.524} C_VEL
LIN {X 0,Y 460.546,Z 277.425,A -85,B 0,C 180,E1 -8065.624,E2 -8065.624} C_VEL
LIN {X 0,Y 460.537,Z 277.429,A -85,B 0,C 180,E1 -8068.745,E2 -8068.745} C_VEL
LIN {X 0,Y 460.582,Z 277.409,A -85,B 0,C 180,E1 -8072.254,E2 -8072.254} C_VEL
LIN {X 0,Y 460.56,Z 277.431,A -85,B 0,C 180,E1 -8074.706,E2 -8074.706} C_VEL
LIN {X 0,Y 460.512,Z 277.419,A -85,B 0,C 180,E1 -8077.572,E2 -8077.572} C_VEL
LIN {X 0,Y 460.57,Z 277.427,A -85,B 0,C 180,E1 -8080.385,E2 -8080.385} C_VEL
LIN {X 0,Y 460.565,Z 277.411,A -85,B 0,C 180,E1 -8083.147,E2 -8083.147} C_VEL
LIN {X 0,Y 460.554,Z 277.426,A -85,B 0,C 180,E1 -8085.868,E2 -8085.868} C_VEL
LIN {X 0,Y 460.611,Z 277.408,A -85,B 0,C 180,E1 -8088.56,E2 -8088.56} C_VEL
LIN {X 0,Y 460.619,Z 277.417,A -85,B 0,C 180,E1 -8091.224,E2 -8091.224} C_VEL
LIN {X 0,Y 460.679,Z 277.409,A -85,B 0,C 180,E1 -8093.87,E2 -8093.87} C_VEL
LIN {X 0,Y 460.793,Z 277.393,A -85,B 0,C 180,E1 -8097.378,E2 -8097.378} C_VEL
LIN {X 0,Y 460.85,Z 277.391,A -85,B 0,C 180,E1 -8100,E2 -8100} C_VEL
LIN {X 0,Y 460.761,Z 277.389,A -85,B 0,C 180,E1 -8102.623,E2 -8102.623} C_VEL
LIN {X 0,Y 460.677,Z 277.414,A -85,B 0,C 180,E1 -8106.131,E2 -8106.131} C_VEL
LIN {X 0,Y 460.611,Z 277.411,A -85,B 0,C 180,E1 -8108.777,E2 -8108.777} C_VEL
LIN {X 0,Y 460.612,Z 277.416,A -85,B 0,C 180,E1 -8112.335,E2 -8112.335} C_VEL
LIN {X 0,Y 460.56,Z 277.426,A -85,B 0,C 180,E1 -8115.979,E2 -8115.979} C_VEL
LIN {X 0,Y 460.568,Z 277.412,A -85,B 0,C 180,E1 -8119.616,E2 -8119.616} C_VEL
LIN {X 0,Y 460.5,Z 277.432,A -85,B 0,C 180,E1 -8122.43,E2 -8122.43} C_VEL
LIN {X 0,Y 460.524,Z 277.432,A -85,B 0,C 180,E1 -8125.79,E2 -8125.79} C_VEL
LIN {X 0,Y 460.498,Z 277.427,A -85,B 0,C 180,E1 -8128.237,E2 -8128.237} C_VEL
LIN {X 0,Y 460.498,Z 277.433,A -85,B 0,C 180,E1 -8131.278,E2 -8131.278} C_VEL
LIN {X 0,Y 460.51,Z 277.433,A -85,B 0,C 180,E1 -8134.501,E2 -8134.501} C_VEL
LIN {X 0,Y 460.481,Z 277.441,A -85,B 0,C 180,E1 -8137.626,E2 -8137.626} C_VEL
LIN {X 0,Y 460.502,Z 277.431,A -85,B 0,C 180,E1 -8141.015,E2 -8141.015} C_VEL
LIN {X 0,Y 460.511,Z 277.434,A -85,B 0,C 180,E1 -8144.59,E2 -8144.59} C_VEL
LIN {X 0,Y 460.544,Z 277.539,A -85,B 0,C 180,E1 -8145.56,E2 -8145.56} C_VEL
LIN {X 0,Y 463.365,Z 286.465,A -85,B 0,C 180,E1 -8146.969,E2 -8146.969} C_VEL
LIN {X 0,Y 472.469,Z 304.698,A -85,B 0,C 180,E1 -8147.99,E2 -8147.99} C_VEL
LIN {X 0,Y 474.576,Z 309.422,A -85,B 0,C 180,E1 -8148.227,E2 -8148.227} C_VEL
LIN {X 0,Y 471.562,Z 491.865,A -85,B 0,C 180,E1 -8151.181,E2 -8151.181} C_VEL
LIN {X 0,Y 471.06,Z 504.923,A -85,B 0,C 180,E1 -8151.512,E2 -8151.512} C_VEL
LIN {X 0,Y 469.495,Z 512.538,A -85,B 0,C 180,E1 -8151.675,E2 -8151.675} C_VEL
LIN {X 0,Y 466.942,Z 519.987,A -85,B 0,C 180,E1 -8151.809,E2 -8151.809} C_VEL
LIN {X 0,Y 464.067,Z 529.235,A -85,B 0,C 180,E1 -8152.061,E2 -8152.061} C_VEL
LIN {X 0,Y 463.128,Z 534.7,A -85,B 0,C 180,E1 -8152.297,E2 -8152.297} C_VEL
LIN {X 0,Y 461.966,Z 550.426,A -85,B 0,C 180,E1 -8153.2,E2 -8153.2} C_VEL
LIN {X 0,Y 460.698,Z 565.582,A -85,B 0,C 180,E1 -8154.275,E2 -8154.275} C_VEL
LIN {X 0,Y 459.495,Z 578.85,A -85,B 0,C 180,E1 -8155.401,E2 -8155.401} C_VEL
LIN {X 0,Y 458.165,Z 592.132,A -85,B 0,C 180,E1 -8156.744,E2 -8156.744} C_VEL
LIN {X 0,Y 456.919,Z 604.644,A -85,B 0,C 180,E1 -8158.244,E2 -8158.244} C_VEL
LIN {X 0,Y 455.835,Z 615.664,A -85,B 0,C 180,E1 -8159.797,E2 -8159.797} C_VEL
LIN {X 0,Y 454.958,Z 625.341,A -85,B 0,C 180,E1 -8161.388,E2 -8161.388} C_VEL
LIN {X 0,Y 454.089,Z 635.275,A -85,B 0,C 180,E1 -8163.331,E2 -8163.331} C_VEL
LIN {X 0,Y 453.441,Z 643.401,A -85,B 0,C 180,E1 -8165.261,E2 -8165.261} C_VEL
LIN {X 0,Y 453.004,Z 650.002,A -85,B 0,C 180,E1 -8167.179,E2 -8167.179} C_VEL
LIN {X 0,Y 452.734,Z 655.284,A -85,B 0,C 180,E1 -8169.081,E2 -8169.081} C_VEL
LIN {X 0,Y 452.523,Z 659.324,A -85,B 0,C 180,E1 -8170.965,E2 -8170.965} C_VEL
LIN {X 0,Y 452.356,Z 662.173,A -85,B 0,C 180,E1 -8172.831,E2 -8172.831} C_VEL
LIN {X 0,Y 452.37,Z 664.023,A -85,B 0,C 180,E1 -8174.686,E2 -8174.686} C_VEL
LIN {X 0,Y 452.34,Z 664.753,A -85,B 0,C 180,E1 -8176.523,E2 -8176.523} C_VEL
LIN {X 0,Y 452.46,Z 664.559,A -85,B 0,C 180,E1 -8178.35,E2 -8178.35} C_VEL
LIN {X 0,Y 452.359,Z 663.331,A -85,B 0,C 180,E1 -8180.16,E2 -8180.16} C_VEL
LIN {X 0,Y 452.446,Z 661.169,A -85,B 0,C 180,E1 -8181.964,E2 -8181.964} C_VEL
LIN {X 0,Y 452.636,Z 657.965,A -85,B 0,C 180,E1 -8183.76,E2 -8183.76} C_VEL
LIN {X 0,Y 452.753,Z 653.765,A -85,B 0,C 180,E1 -8185.548,E2 -8185.548} C_VEL
LIN {X 0,Y 452.997,Z 648.493,A -85,B 0,C 180,E1 -8187.332,E2 -8187.332} C_VEL
LIN {X 0,Y 453.494,Z 641.998,A -85,B 0,C 180,E1 -8189.112,E2 -8189.112} C_VEL
LIN {X 0,Y 454.057,Z 633.193,A -85,B 0,C 180,E1 -8191.109,E2 -8191.109} C_VEL
LIN {X 0,Y 454.907,Z 623.792,A -85,B 0,C 180,E1 -8192.878,E2 -8192.878} C_VEL
LIN {X 0,Y 456.001,Z 612.627,A -85,B 0,C 180,E1 -8194.641,E2 -8194.641} C_VEL
LIN {X 0,Y 457.067,Z 601.061,A -85,B 0,C 180,E1 -8196.179,E2 -8196.179} C_VEL
LIN {X 0,Y 458.162,Z 588.458,A -85,B 0,C 180,E1 -8197.603,E2 -8197.603} C_VEL
LIN {X 0,Y 459.446,Z 574.708,A -85,B 0,C 180,E1 -8198.91,E2 -8198.91} C_VEL
LIN {X 0,Y 460.559,Z 561.187,A -85,B 0,C 180,E1 -8199.996,E2 -8199.996} C_VEL
LIN {X 0,Y 461.685,Z 546.588,A -85,B 0,C 180,E1 -8200.969,E2 -8200.969} C_VEL
LIN {X 0,Y 462.616,Z 532.633,A -85,B 0,C 180,E1 -8201.724,E2 -8201.724} C_VEL
LIN {X 0,Y 463.409,Z 517.898,A -85,B 0,C 180,E1 -8202.37,E2 -8202.37} C_VEL
LIN {X 0,Y 464.165,Z 501.575,A -85,B 0,C 180,E1 -8202.905,E2 -8202.905} C_VEL
LIN {X 0,Y 464.699,Z 484.172,A -85,B 0,C 180,E1 -8203.279,E2 -8203.279} C_VEL
LIN {X 0,Y 467.373,Z 311.601,A -85,B 0,C 180,E1 -8206.039,E2 -8206.039} C_VEL
LIN {X 0,Y 466.752,Z 309.564,A -85,B 0,C 180,E1 -8206.113,E2 -8206.113} C_VEL
LIN {X 0,Y 455.722,Z 285.971,A -85,B 0,C 180,E1 -8207.261,E2 -8207.261} C_VEL
LIN {X 0,Y 453.55,Z 278.302,A -85,B 0,C 180,E1 -8208.404,E2 -8208.404} C_VEL
LIN {X 0,Y 453.48,Z 278.303,A -85,B 0,C 180,E1 -8211.836,E2 -8211.836} C_VEL
LIN {X 0,Y 453.467,Z 278.31,A -85,B 0,C 180,E1 -8214.737,E2 -8214.737} C_VEL
LIN {X 0,Y 453.462,Z 278.316,A -85,B 0,C 180,E1 -8217.942,E2 -8217.942} C_VEL
LIN {X 0,Y 453.457,Z 278.313,A -85,B 0,C 180,E1 -8220.761,E2 -8220.761} C_VEL
LIN {X 0,Y 453.455,Z 278.317,A -85,B 0,C 180,E1 -8223.914,E2 -8223.914} C_VEL
LIN {X 0,Y 453.431,Z 278.313,A -85,B 0,C 180,E1 -8227.192,E2 -8227.192} C_VEL
LIN {X 0,Y 453.466,Z 278.309,A -85,B 0,C 180,E1 -8230.612,E2 -8230.612} C_VEL
LIN {X 0,Y 453.477,Z 278.308,A -85,B 0,C 180,E1 -8234.527,E2 -8234.527} C_VEL
LIN {X 0,Y 453.433,Z 278.318,A -85,B 0,C 180,E1 -8238.071,E2 -8238.071} C_VEL
LIN {X 0,Y 453.431,Z 278.307,A -85,B 0,C 180,E1 -8240.803,E2 -8240.803} C_VEL
LIN {X 0,Y 453.442,Z 278.288,A -85,B 0,C 180,E1 -8243.915,E2 -8243.915} C_VEL
LIN {X 0,Y 453.475,Z 278.306,A -85,B 0,C 180,E1 -8247.15,E2 -8247.15} C_VEL
LIN {X 0,Y 453.462,Z 278.302,A -85,B 0,C 180,E1 -8250.267,E2 -8250.267} C_VEL
LIN {X 0,Y 453.441,Z 278.313,A -85,B 0,C 180,E1 -8253.289,E2 -8253.289} C_VEL
LIN {X 0,Y 453.494,Z 278.299,A -85,B 0,C 180,E1 -8256.238,E2 -8256.238} C_VEL
LIN {X 0,Y 453.484,Z 278.308,A -85,B 0,C 180,E1 -8259.117,E2 -8259.117} C_VEL
LIN {X 0,Y 453.502,Z 278.299,A -85,B 0,C 180,E1 -8261.944,E2 -8261.944} C_VEL
LIN {X 0,Y 453.539,Z 278.299,A -85,B 0,C 180,E1 -8264.726,E2 -8264.726} C_VEL
LIN {X 0,Y 453.56,Z 278.289,A -85,B 0,C 180,E1 -8268.378,E2 -8268.378} C_VEL
LIN {X 0,Y 453.585,Z 278.296,A -85,B 0,C 180,E1 -8271.086,E2 -8271.086} C_VEL
LIN {X 0,Y 453.669,Z 278.277,A -85,B 0,C 180,E1 -8273.774,E2 -8273.774} C_VEL
LIN {X 0,Y 453.733,Z 278.281,A -85,B 0,C 180,E1 -8277.336,E2 -8277.336} C_VEL
LIN {X 0,Y 453.822,Z 278.255,A -85,B 0,C 180,E1 -8280,E2 -8280} C_VEL
LIN {X 0,Y 453.744,Z 278.273,A -85,B 0,C 180,E1 -8282.663,E2 -8282.663} C_VEL
LIN {X 0,Y 453.653,Z 278.275,A -85,B 0,C 180,E1 -8286.225,E2 -8286.225} C_VEL
LIN {X 0,Y 453.592,Z 278.289,A -85,B 0,C 180,E1 -8288.913,E2 -8288.913} C_VEL
LIN {X 0,Y 453.564,Z 278.294,A -85,B 0,C 180,E1 -8292.528,E2 -8292.528} C_VEL
LIN {X 0,Y 453.544,Z 278.297,A -85,B 0,C 180,E1 -8296.195,E2 -8296.195} C_VEL
LIN {X 0,Y 453.517,Z 278.307,A -85,B 0,C 180,E1 -8299.039,E2 -8299.039} C_VEL
LIN {X 0,Y 453.476,Z 278.307,A -85,B 0,C 180,E1 -8301.836,E2 -8301.836} C_VEL
LIN {X 0,Y 453.514,Z 278.307,A -85,B 0,C 180,E1 -8304.734,E2 -8304.734} C_VEL
LIN {X 0,Y 453.531,Z 278.299,A -85,B 0,C 180,E1 -8307.959,E2 -8307.959} C_VEL
LIN {X 0,Y 453.465,Z 278.312,A -85,B 0,C 180,E1 -8311.525,E2 -8311.525} C_VEL
LIN {X 0,Y 453.488,Z 278.311,A -85,B 0,C 180,E1 -8314.777,E2 -8314.777} C_VEL
LIN {X 0,Y 453.472,Z 278.308,A -85,B 0,C 180,E1 -8318.31,E2 -8318.31} C_VEL
LIN {X 0,Y 453.493,Z 278.305,A -85,B 0,C 180,E1 -8320.609,E2 -8320.609} C_VEL
LIN {X 0,Y 453.463,Z 278.311,A -85,B 0,C 180,E1 -8323.245,E2 -8323.245} C_VEL
LIN {X 0,Y 453.472,Z 278.31,A -85,B 0,C 180,E1 -8325.78,E2 -8325.78} C_VEL
LIN {X 0,Y 453.48,Z 278.307,A -85,B 0,C 180,E1 -8328.209,E2 -8328.209} C_VEL
LIN {X 0,Y 453.514,Z 278.308,A -85,B 0,C 180,E1 -8330.79,E2 -8330.79} C_VEL
LIN {X 0,Y 453.452,Z 278.312,A -85,B 0,C 180,E1 -8333.917,E2 -8333.917} C_VEL
LIN {X 0,Y 453.567,Z 278.491,A -85,B 0,C 180,E1 -8336.144,E2 -8336.144} C_VEL
LIN {X 0,Y 460.453,Z 301.064,A -85,B 0,C 180,E1 -8339.21,E2 -8339.21} C_VEL
LIN {X 0,Y 462.397,Z 308.504,A -85,B 0,C 180,E1 -8340.165,E2 -8340.165} C_VEL
LIN {X 0,Y 462.429,Z 309.639,A -85,B 0,C 180,E1 -8340.236,E2 -8340.236} C_VEL
LIN {X 0,Y 467.16,Z 337.267,A -85,B 0,C 180,E1 -8341.009,E2 -8341.009} C_VEL
LIN {X 0,Y 464.409,Z 514.191,A -85,B 0,C 180,E1 -8343.849,E2 -8343.849} C_VEL
LIN {X 0,Y 463.756,Z 530.899,A -85,B 0,C 180,E1 -8344.261,E2 -8344.261} C_VEL
LIN {X 0,Y 462.94,Z 547.306,A -85,B 0,C 180,E1 -8344.845,E2 -8344.845} C_VEL
LIN {X 0,Y 461.935,Z 562.834,A -85,B 0,C 180,E1 -8345.567,E2 -8345.567} C_VEL
LIN {X 0,Y 460.859,Z 577.342,A -85,B 0,C 180,E1 -8346.419,E2 -8346.419} C_VEL
LIN {X 0,Y 459.656,Z 591.305,A -85,B 0,C 180,E1 -8347.409,E2 -8347.409} C_VEL
LIN {X 0,Y 458.49,Z 604.654,A -85,B 0,C 180,E1 -8348.533,E2 -8348.533} C_VEL
LIN {X 0,Y 457.287,Z 618.389,A -85,B 0,C 180,E1 -8349.908,E2 -8349.908} C_VEL
LIN {X 0,Y 456.169,Z 630.561,A -85,B 0,C 180,E1 -8351.356,E2 -8351.356} C_VEL
LIN {X 0,Y 455.162,Z 641.901,A -85,B 0,C 180,E1 -8352.94,E2 -8352.94} C_VEL
LIN {X 0,Y 454.285,Z 652.875,A -85,B 0,C 180,E1 -8354.752,E2 -8354.752} C_VEL
LIN {X 0,Y 453.604,Z 662.086,A -85,B 0,C 180,E1 -8356.561,E2 -8356.561} C_VEL
LIN {X 0,Y 453.156,Z 669.786,A -85,B 0,C 180,E1 -8358.369,E2 -8358.369} C_VEL
LIN {X 0,Y 452.723,Z 677.517,A -85,B 0,C 180,E1 -8360.619,E2 -8360.619} C_VEL
LIN {X 0,Y 452.569,Z 683.391,A -85,B 0,C 180,E1 -8362.864,E2 -8362.864} C_VEL
LIN {X 0,Y 452.495,Z 686.827,A -85,B 0,C 180,E1 -8364.653,E2 -8364.653} C_VEL
LIN {X 0,Y 452.456,Z 689.321,A -85,B 0,C 180,E1 -8366.438,E2 -8366.438} C_VEL
LIN {X 0,Y 452.427,Z 690.726,A -85,B 0,C 180,E1 -8368.22,E2 -8368.22} C_VEL
LIN {X 0,Y 452.429,Z 691.253,A -85,B 0,C 180,E1 -8370,E2 -8370} C_VEL
LIN {X 0,Y 452.447,Z 690.72,A -85,B 0,C 180,E1 -8371.78,E2 -8371.78} C_VEL
LIN {X 0,Y 452.456,Z 689.309,A -85,B 0,C 180,E1 -8373.562,E2 -8373.562} C_VEL
LIN {X 0,Y 452.495,Z 686.815,A -85,B 0,C 180,E1 -8375.347,E2 -8375.347} C_VEL
LIN {X 0,Y 452.569,Z 683.389,A -85,B 0,C 180,E1 -8377.137,E2 -8377.137} C_VEL
LIN {X 0,Y 452.723,Z 677.532,A -85,B 0,C 180,E1 -8379.381,E2 -8379.381} C_VEL
LIN {X 0,Y 453.156,Z 669.844,A -85,B 0,C 180,E1 -8381.632,E2 -8381.632} C_VEL
LIN {X 0,Y 453.663,Z 661.175,A -85,B 0,C 180,E1 -8383.665,E2 -8383.665} C_VEL
LIN {X 0,Y 454.422,Z 651.839,A -85,B 0,C 180,E1 -8385.473,E2 -8385.473} C_VEL
LIN {X 0,Y 455.224,Z 642.259,A -85,B 0,C 180,E1 -8387.058,E2 -8387.058} C_VEL
LIN {X 0,Y 456.258,Z 631.123,A -85,B 0,C 180,E1 -8388.64,E2 -8388.64} C_VEL
LIN {X 0,Y 457.501,Z 618.05,A -85,B 0,C 180,E1 -8390.213,E2 -8390.213} C_VEL
LIN {X 0,Y 458.743,Z 604.597,A -85,B 0,C 180,E1 -8391.573,E2 -8391.573} C_VEL
LIN {X 0,Y 459.923,Z 591.442,A -85,B 0,C 180,E1 -8392.696,E2 -8392.696} C_VEL
LIN {X 0,Y 461.292,Z 576.179,A -85,B 0,C 180,E1 -8393.784,E2 -8393.784} C_VEL
LIN {X 0,Y 462.555,Z 560.409,A -85,B 0,C 180,E1 -8394.698,E2 -8394.698} C_VEL
LIN {X 0,Y 463.622,Z 544.719,A -85,B 0,C 180,E1 -8395.416,E2 -8395.416} C_VEL
LIN {X 0,Y 464.448,Z 528.571,A -85,B 0,C 180,E1 -8395.969,E2 -8395.969} C_VEL
LIN {X 0,Y 465.096,Z 512.515,A -85,B 0,C 180,E1 -8396.348,E2 -8396.348} C_VEL
LIN {X 0,Y 468.128,Z 337.473,A -85,B 0,C 180,E1 -8399.205,E2 -8399.205} C_VEL
LIN {X 0,Y 464.331,Z 315.005,A -85,B 0,C 180,E1 -8399.89,E2 -8399.89} C_VEL
LIN {X 0,Y 462.981,Z 308.562,A -85,B 0,C 180,E1 -8400.122,E2 -8400.122} C_VEL
LIN {X 0,Y 458.583,Z 293.486,A -85,B 0,C 180,E1 -8402.251,E2 -8402.251} C_VEL
LIN {X 0,Y 454.42,Z 280.999,A -85,B 0,C 180,E1 -8404.143,E2 -8404.143} C_VEL
LIN {X 0,Y 453.494,Z 278.306,A -85,B 0,C 180,E1 -8404.582,E2 -8404.582} C_VEL
LIN {X 0,Y 453.471,Z 278.314,A -85,B 0,C 180,E1 -8407.777,E2 -8407.777} C_VEL
LIN {X 0,Y 453.493,Z 278.31,A -85,B 0,C 180,E1 -8410.609,E2 -8410.609} C_VEL
LIN {X 0,Y 453.463,Z 278.314,A -85,B 0,C 180,E1 -8413.246,E2 -8413.246} C_VEL
LIN {X 0,Y 453.466,Z 278.308,A -85,B 0,C 180,E1 -8415.779,E2 -8415.779} C_VEL
LIN {X 0,Y 453.479,Z 278.303,A -85,B 0,C 180,E1 -8418.21,E2 -8418.21} C_VEL
LIN {X 0,Y 453.51,Z 278.309,A -85,B 0,C 180,E1 -8420.791,E2 -8420.791} C_VEL
LIN {X 0,Y 453.454,Z 278.31,A -85,B 0,C 180,E1 -8423.918,E2 -8423.918} C_VEL
LIN {X 0,Y 453.483,Z 278.299,A -85,B 0,C 180,E1 -8427.152,E2 -8427.152} C_VEL
LIN {X 0,Y 453.475,Z 278.309,A -85,B 0,C 180,E1 -8430.269,E2 -8430.269} C_VEL
LIN {X 0,Y 453.508,Z 278.304,A -85,B 0,C 180,E1 -8433.294,E2 -8433.294} C_VEL
LIN {X 0,Y 453.505,Z 278.301,A -85,B 0,C 180,E1 -8436.239,E2 -8436.239} C_VEL
LIN {X 0,Y 453.484,Z 278.309,A -85,B 0,C 180,E1 -8439.118,E2 -8439.118} C_VEL
LIN {X 0,Y 453.512,Z 278.299,A -85,B 0,C 180,E1 -8441.945,E2 -8441.945} C_VEL
LIN {X 0,Y 453.541,Z 278.295,A -85,B 0,C 180,E1 -8444.727,E2 -8444.727} C_VEL
LIN {X 0,Y 453.56,Z 278.288,A -85,B 0,C 180,E1 -8448.379,E2 -8448.379} C_VEL
LIN {X 0,Y 453.585,Z 278.295,A -85,B 0,C 180,E1 -8451.087,E2 -8451.087} C_VEL
LIN {X 0,Y 453.646,Z 278.285,A -85,B 0,C 180,E1 -8453.775,E2 -8453.775} C_VEL
LIN {X 0,Y 453.737,Z 278.272,A -85,B 0,C 180,E1 -8457.337,E2 -8457.337} C_VEL
LIN {X 0,Y 453.82,Z 278.267,A -85,B 0,C 180,E1 -8460,E2 -8460} C_VEL
LIN {X 0,Y 453.708,Z 278.268,A -85,B 0,C 180,E1 -8462.664,E2 -8462.664} C_VEL
LIN {X 0,Y 453.644,Z 278.287,A -85,B 0,C 180,E1 -8466.226,E2 -8466.226} C_VEL
LIN {X 0,Y 453.579,Z 278.287,A -85,B 0,C 180,E1 -8468.914,E2 -8468.914} C_VEL
LIN {X 0,Y 453.567,Z 278.29,A -85,B 0,C 180,E1 -8472.529,E2 -8472.529} C_VEL
LIN {X 0,Y 453.506,Z 278.306,A -85,B 0,C 180,E1 -8476.092,E2 -8476.092} C_VEL
LIN {X 0,Y 453.52,Z 278.288,A -85,B 0,C 180,E1 -8479.04,E2 -8479.04} C_VEL
LIN {X 0,Y 453.476,Z 278.312,A -85,B 0,C 180,E1 -8481.837,E2 -8481.837} C_VEL
LIN {X 0,Y 453.464,Z 278.307,A -85,B 0,C 180,E1 -8484.738,E2 -8484.738} C_VEL
LIN {X 0,Y 453.458,Z 278.305,A -85,B 0,C 180,E1 -8487.941,E2 -8487.941} C_VEL
LIN {X 0,Y 453.449,Z 278.312,A -85,B 0,C 180,E1 -8490.762,E2 -8490.762} C_VEL
LIN {X 0,Y 453.455,Z 278.318,A -85,B 0,C 180,E1 -8493.915,E2 -8493.915} C_VEL
LIN {X 0,Y 453.433,Z 278.318,A -85,B 0,C 180,E1 -8497.192,E2 -8497.192} C_VEL
LIN {X 0,Y 453.467,Z 278.309,A -85,B 0,C 180,E1 -8500.613,E2 -8500.613} C_VEL
LIN {X 0,Y 453.481,Z 278.311,A -85,B 0,C 180,E1 -8504.528,E2 -8504.528} C_VEL
LIN {X 0,Y 453.465,Z 278.31,A -85,B 0,C 180,E1 -8505.026,E2 -8505.026} C_VEL
LIN {X 0,Y 456.181,Z 286.803,A -85,B 0,C 180,E1 -8506.394,E2 -8506.394} C_VEL
LIN {X 0,Y 464.708,Z 303.346,A -85,B 0,C 180,E1 -8507.38,E2 -8507.38} C_VEL
LIN {X 0,Y 468.413,Z 311.369,A -85,B 0,C 180,E1 -8507.806,E2 -8507.806} C_VEL
LIN {X 0,Y 465.738,Z 465.13,A -85,B 0,C 180,E1 -8510.312,E2 -8510.312} C_VEL
LIN {X 0,Y 465.186,Z 494.274,A -85,B 0,C 180,E1 -8510.824,E2 -8510.824} C_VEL
LIN {X 0,Y 464.449,Z 511.524,A -85,B 0,C 180,E1 -8511.308,E2 -8511.308} C_VEL
LIN {X 0,Y 463.658,Z 526.679,A -85,B 0,C 180,E1 -8511.912,E2 -8511.912} C_VEL
LIN {X 0,Y 463.128,Z 534.7,A -85,B 0,C 180,E1 -8512.297,E2 -8512.297} C_VEL
LIN {X 0,Y 462.09,Z 540.194,A -85,B 0,C 180,E1 -8512.543,E2 -8512.543} C_VEL
LIN {X 0,Y 456.074,Z 556.052,A -85,B 0,C 180,E1 -8513.234,E2 -8513.234} C_VEL
LIN {X 0,Y 454.709,Z 561.202,A -85,B 0,C 180,E1 -8513.548,E2 -8513.548} C_VEL
LIN {X 0,Y 454.489,Z 562.892,A -85,B 0,C 180,E1 -8513.67,E2 -8513.67} C_VEL
LIN {X 0,Y 453.13,Z 576.887,A -85,B 0,C 180,E1 -8514.844,E2 -8514.844} C_VEL
LIN {X 0,Y 451.722,Z 590.502,A -85,B 0,C 180,E1 -8516.206,E2 -8516.206} C_VEL
LIN {X 0,Y 450.297,Z 603.679,A -85,B 0,C 180,E1 -8517.774,E2 -8517.774} C_VEL
LIN {X 0,Y 449.098,Z 615.184,A -85,B 0,C 180,E1 -8519.397,E2 -8519.397} C_VEL
LIN {X 0,Y 448.209,Z 624.409,A -85,B 0,C 180,E1 -8520.916,E2 -8520.916} C_VEL
LIN {X 0,Y 447.333,Z 633.333,A -85,B 0,C 180,E1 -8522.642,E2 -8522.642} C_VEL
LIN {X 0,Y 446.69,Z 640.913,A -85,B 0,C 180,E1 -8524.363,E2 -8524.363} C_VEL
LIN {X 0,Y 446.109,Z 648.349,A -85,B 0,C 180,E1 -8526.399,E2 -8526.399} C_VEL
LIN {X 0,Y 445.704,Z 655.024,A -85,B 0,C 180,E1 -8528.736,E2 -8528.736} C_VEL
LIN {X 0,Y 445.46,Z 659.141,A -85,B 0,C 180,E1 -8530.651,E2 -8530.651} C_VEL
LIN {X 0,Y 445.273,Z 662.137,A -85,B 0,C 180,E1 -8532.549,E2 -8532.549} C_VEL
LIN {X 0,Y 445.297,Z 664.07,A -85,B 0,C 180,E1 -8534.436,E2 -8534.436} C_VEL
LIN {X 0,Y 445.249,Z 664.927,A -85,B 0,C 180,E1 -8536.304,E2 -8536.304} C_VEL
LIN {X 0,Y 445.39,Z 664.843,A -85,B 0,C 180,E1 -8538.163,E2 -8538.163} C_VEL
LIN {X 0,Y 445.284,Z 663.708,A -85,B 0,C 180,E1 -8540.002,E2 -8540.002} C_VEL
LIN {X 0,Y 445.342,Z 661.677,A -85,B 0,C 180,E1 -8541.835,E2 -8541.835} C_VEL
LIN {X 0,Y 445.533,Z 658.549,A -85,B 0,C 180,E1 -8543.66,E2 -8543.66} C_VEL
LIN {X 0,Y 445.655,Z 654.49,A -85,B 0,C 180,E1 -8545.477,E2 -8545.477} C_VEL
LIN {X 0,Y 445.927,Z 649.287,A -85,B 0,C 180,E1 -8547.29,E2 -8547.29} C_VEL
LIN {X 0,Y 446.43,Z 642.944,A -85,B 0,C 180,E1 -8549.098,E2 -8549.098} C_VEL
LIN {X 0,Y 446.958,Z 635.381,A -85,B 0,C 180,E1 -8550.901,E2 -8550.901} C_VEL
LIN {X 0,Y 447.785,Z 626.271,A -85,B 0,C 180,E1 -8552.699,E2 -8552.699} C_VEL
LIN {X 0,Y 448.719,Z 616.936,A -85,B 0,C 180,E1 -8554.266,E2 -8554.266} C_VEL
LIN {X 0,Y 449.772,Z 606.134,A -85,B 0,C 180,E1 -8555.829,E2 -8555.829} C_VEL
LIN {X 0,Y 450.978,Z 593.43,A -85,B 0,C 180,E1 -8557.387,E2 -8557.387} C_VEL
LIN {X 0,Y 452.219,Z 580.505,A -85,B 0,C 180,E1 -8558.715,E2 -8558.715} C_VEL
LIN {X 0,Y 453.469,Z 566.517,A -85,B 0,C 180,E1 -8559.928,E2 -8559.928} C_VEL
LIN {X 0,Y 454.778,Z 551.199,A -85,B 0,C 180,E1 -8561.025,E2 -8561.025} C_VEL
LIN {X 0,Y 455.805,Z 536.285,A -85,B 0,C 180,E1 -8561.901,E2 -8561.901} C_VEL
LIN {X 0,Y 456.813,Z 520.991,A -85,B 0,C 180,E1 -8562.608,E2 -8562.608} C_VEL
LIN {X 0,Y 457.571,Z 504.63,A -85,B 0,C 180,E1 -8563.179,E2 -8563.179} C_VEL
LIN {X 0,Y 458.162,Z 487.55,A -85,B 0,C 180,E1 -8563.585,E2 -8563.585} C_VEL
LIN {X 0,Y 461.044,Z 312.986,A -85,B 0,C 180,E1 -8566.42,E2 -8566.42} C_VEL
LIN {X 0,Y 448.496,Z 286.177,A -85,B 0,C 180,E1 -8567.751,E2 -8567.751} C_VEL
LIN {X 0,Y 446.498,Z 279.181,A -85,B 0,C 180,E1 -8568.825,E2 -8568.825} C_VEL
LIN {X 0,Y 446.42,Z 279.182,A -85,B 0,C 180,E1 -8572.199,E2 -8572.199} C_VEL
LIN {X 0,Y 446.417,Z 279.186,A -85,B 0,C 180,E1 -8575.155,E2 -8575.155} C_VEL
LIN {X 0,Y 446.419,Z 279.196,A -85,B 0,C 180,E1 -8578.183,E2 -8578.183} C_VEL
LIN {X 0,Y 446.394,Z 279.193,A -85,B 0,C 180,E1 -8581.302,E2 -8581.302} C_VEL
LIN {X 0,Y 446.413,Z 279.185,A -85,B 0,C 180,E1 -8584.524,E2 -8584.524} C_VEL
LIN {X 0,Y 446.386,Z 279.192,A -85,B 0,C 180,E1 -8587.881,E2 -8587.881} C_VEL
LIN {X 0,Y 446.396,Z 279.188,A -85,B 0,C 180,E1 -8590.912,E2 -8590.912} C_VEL
LIN {X 0,Y 446.384,Z 279.195,A -85,B 0,C 180,E1 -8593.848,E2 -8593.848} C_VEL
LIN {X 0,Y 446.381,Z 279.187,A -85,B 0,C 180,E1 -8596.406,E2 -8596.406} C_VEL
LIN {X 0,Y 446.393,Z 279.193,A -85,B 0,C 180,E1 -8599.796,E2 -8599.796} C_VEL
LIN {X 0,Y 446.393,Z 279.162,A -85,B 0,C 180,E1 -8603.253,E2 -8603.253} C_VEL
LIN {X 0,Y 446.451,Z 279.18,A -85,B 0,C 180,E1 -8606.566,E2 -8606.566} C_VEL
LIN {X 0,Y 446.428,Z 279.181,A -85,B 0,C 180,E1 -8609.98,E2 -8609.98} C_VEL
LIN {X 0,Y 446.394,Z 279.189,A -85,B 0,C 180,E1 -8612.833,E2 -8612.833} C_VEL
LIN {X 0,Y 446.425,Z 279.18,A -85,B 0,C 180,E1 -8615.935,E2 -8615.935} C_VEL
LIN {X 0,Y 446.455,Z 279.182,A -85,B 0,C 180,E1 -8618.773,E2 -8618.773} C_VEL
LIN {X 0,Y 446.452,Z 279.178,A -85,B 0,C 180,E1 -8621.648,E2 -8621.648} C_VEL
LIN {X 0,Y 446.508,Z 279.175,A -85,B 0,C 180,E1 -8624.479,E2 -8624.479} C_VEL
LIN {X 0,Y 446.518,Z 279.166,A -85,B 0,C 180,E1 -8628.193,E2 -8628.193} C_VEL
LIN {X 0,Y 446.532,Z 279.173,A -85,B 0,C 180,E1 -8630.944,E2 -8630.944} C_VEL
LIN {X 0,Y 446.638,Z 279.153,A -85,B 0,C 180,E1 -8633.676,E2 -8633.676} C_VEL
LIN {X 0,Y 446.68,Z 279.159,A -85,B 0,C 180,E1 -8637.294,E2 -8637.294} C_VEL
LIN {X 0,Y 446.792,Z 279.13,A -85,B 0,C 180,E1 -8640,E2 -8640} C_VEL
LIN {X 0,Y 446.691,Z 279.152,A -85,B 0,C 180,E1 -8642.705,E2 -8642.705} C_VEL
LIN {X 0,Y 446.621,Z 279.15,A -85,B 0,C 180,E1 -8646.324,E2 -8646.324} C_VEL
LIN {X 0,Y 446.538,Z 279.169,A -85,B 0,C 180,E1 -8649.055,E2 -8649.055} C_VEL
LIN {X 0,Y 446.521,Z 279.172,A -85,B 0,C 180,E1 -8652.729,E2 -8652.729} C_VEL
LIN {X 0,Y 446.495,Z 279.175,A -85,B 0,C 180,E1 -8656.227,E2 -8656.227} C_VEL
LIN {X 0,Y 446.468,Z 279.185,A -85,B 0,C 180,E1 -8659.303,E2 -8659.303} C_VEL
LIN {X 0,Y 446.418,Z 279.185,A -85,B 0,C 180,E1 -8662.199,E2 -8662.199} C_VEL
LIN {X 0,Y 446.457,Z 279.186,A -85,B 0,C 180,E1 -8665.152,E2 -8665.152} C_VEL
LIN {X 0,Y 446.484,Z 279.177,A -85,B 0,C 180,E1 -8668.178,E2 -8668.178} C_VEL
LIN {X 0,Y 446.418,Z 279.188,A -85,B 0,C 180,E1 -8671.775,E2 -8671.775} C_VEL
LIN {X 0,Y 446.429,Z 279.188,A -85,B 0,C 180,E1 -8674.523,E2 -8674.523} C_VEL
LIN {X 0,Y 446.429,Z 279.185,A -85,B 0,C 180,E1 -8678.082,E2 -8678.082} C_VEL
LIN {X 0,Y 446.426,Z 279.184,A -85,B 0,C 180,E1 -8680.917,E2 -8680.917} C_VEL
LIN {X 0,Y 446.422,Z 279.185,A -85,B 0,C 180,E1 -8683.843,E2 -8683.843} C_VEL
LIN {X 0,Y 446.419,Z 279.191,A -85,B 0,C 180,E1 -8686.4,E2 -8686.4} C_VEL
LIN {X 0,Y 446.449,Z 279.185,A -85,B 0,C 180,E1 -8689.803,E2 -8689.803} C_VEL
LIN {X 0,Y 446.407,Z 279.189,A -85,B 0,C 180,E1 -8692.121,E2 -8692.121} C_VEL
LIN {X 0,Y 446.485,Z 279.315,A -85,B 0,C 180,E1 -8695.714,E2 -8695.714} C_VEL
LIN {X 0,Y 453.306,Z 301.512,A -85,B 0,C 180,E1 -8698.793,E2 -8698.793} C_VEL
LIN {X 0,Y 455.505,Z 309.055,A -85,B 0,C 180,E1 -8699.771,E2 -8699.771} C_VEL
LIN {X 0,Y 456.473,Z 312.612,A -85,B 0,C 180,E1 -8699.897,E2 -8699.897} C_VEL
LIN {X 0,Y 460.826,Z 338.425,A -85,B 0,C 180,E1 -8700.63,E2 -8700.63} C_VEL
LIN {X 0,Y 457.905,Z 515.048,A -85,B 0,C 180,E1 -8703.502,E2 -8703.502} C_VEL
LIN {X 0,Y 457.213,Z 531.611,A -85,B 0,C 180,E1 -8703.926,E2 -8703.926} C_VEL
LIN {X 0,Y 456.381,Z 547.784,A -85,B 0,C 180,E1 -8704.518,E2 -8704.518} C_VEL
LIN {X 0,Y 455.334,Z 563.176,A -85,B 0,C 180,E1 -8705.249,E2 -8705.249} C_VEL
LIN {X 0,Y 454.176,Z 578.028,A -85,B 0,C 180,E1 -8706.137,E2 -8706.137} C_VEL
LIN {X 0,Y 452.891,Z 592.24,A -85,B 0,C 180,E1 -8707.173,E2 -8707.173} C_VEL
LIN {X 0,Y 451.657,Z 605.386,A -85,B 0,C 180,E1 -8708.312,E2 -8708.312} C_VEL
LIN {X 0,Y 450.466,Z 618.433,A -85,B 0,C 180,E1 -8709.645,E2 -8709.645} C_VEL
LIN {X 0,Y 449.341,Z 630.169,A -85,B 0,C 180,E1 -8711.062,E2 -8711.062} C_VEL
LIN {X 0,Y 448.261,Z 641.555,A -85,B 0,C 180,E1 -8712.669,E2 -8712.669} C_VEL
LIN {X 0,Y 447.359,Z 652.568,A -85,B 0,C 180,E1 -8714.51,E2 -8714.51} C_VEL
LIN {X 0,Y 446.583,Z 661.804,A -85,B 0,C 180,E1 -8716.346,E2 -8716.346} C_VEL
LIN {X 0,Y 446.127,Z 669.519,A -85,B 0,C 180,E1 -8718.183,E2 -8718.183} C_VEL
LIN {X 0,Y 445.677,Z 675.826,A -85,B 0,C 180,E1 -8720.011,E2 -8720.011} C_VEL
LIN {X 0,Y 445.553,Z 680.998,A -85,B 0,C 180,E1 -8721.839,E2 -8721.839} C_VEL
LIN {X 0,Y 445.486,Z 685.002,A -85,B 0,C 180,E1 -8723.66,E2 -8723.66} C_VEL
LIN {X 0,Y 445.36,Z 687.971,A -85,B 0,C 180,E1 -8725.475,E2 -8725.475} C_VEL
LIN {X 0,Y 445.411,Z 689.922,A -85,B 0,C 180,E1 -8727.287,E2 -8727.287} C_VEL
LIN {X 0,Y 445.334,Z 690.892,A -85,B 0,C 180,E1 -8729.096,E2 -8729.096} C_VEL
LIN {X 0,Y 445.336,Z 690.89,A -85,B 0,C 180,E1 -8730.904,E2 -8730.904} C_VEL
LIN {X 0,Y 445.411,Z 689.929,A -85,B 0,C 180,E1 -8732.713,E2 -8732.713} C_VEL
LIN {X 0,Y 445.36,Z 687.979,A -85,B 0,C 180,E1 -8734.526,E2 -8734.526} C_VEL
LIN {X 0,Y 445.486,Z 685.034,A -85,B 0,C 180,E1 -8736.34,E2 -8736.34} C_VEL
LIN {X 0,Y 445.536,Z 681.048,A -85,B 0,C 180,E1 -8738.162,E2 -8738.162} C_VEL
LIN {X 0,Y 445.681,Z 675.927,A -85,B 0,C 180,E1 -8739.989,E2 -8739.989} C_VEL
LIN {X 0,Y 446.136,Z 669.688,A -85,B 0,C 180,E1 -8741.817,E2 -8741.817} C_VEL
LIN {X 0,Y 446.672,Z 661.039,A -85,B 0,C 180,E1 -8743.883,E2 -8743.883} C_VEL
LIN {X 0,Y 447.504,Z 651.734,A -85,B 0,C 180,E1 -8745.719,E2 -8745.719} C_VEL
LIN {X 0,Y 448.336,Z 642.182,A -85,B 0,C 180,E1 -8747.328,E2 -8747.328} C_VEL
LIN {X 0,Y 449.446,Z 631.073,A -85,B 0,C 180,E1 -8748.933,E2 -8748.933} C_VEL
LIN {X 0,Y 450.796,Z 617.682,A -85,B 0,C 180,E1 -8750.568,E2 -8750.568} C_VEL
LIN {X 0,Y 452.107,Z 604.64,A -85,B 0,C 180,E1 -8751.906,E2 -8751.906} C_VEL
LIN {X 0,Y 453.343,Z 591.574,A -85,B 0,C 180,E1 -8753.044,E2 -8753.044} C_VEL
LIN {X 0,Y 454.741,Z 577.132,A -85,B 0,C 180,E1 -8754.098,E2 -8754.098} C_VEL
LIN {X 0,Y 456.045,Z 561.851,A -85,B 0,C 180,E1 -8755.014,E2 -8755.014} C_VEL
LIN {X 0,Y 457.234,Z 545.148,A -85,B 0,C 180,E1 -8755.797,E2 -8755.797} C_VEL
LIN {X 0,Y 458.122,Z 529.261,A -85,B 0,C 180,E1 -8756.355,E2 -8756.355} C_VEL
LIN {X 0,Y 458.852,Z 512.462,A -85,B 0,C 180,E1 -8756.762,E2 -8756.762} C_VEL
LIN {X 0,Y 462.045,Z 338.71,A -85,B 0,C 180,E1 -8759.639,E2 -8759.639} C_VEL
LIN {X 0,Y 458.305,Z 316.291,A -85,B 0,C 180,E1 -8760.34,E2 -8760.34} C_VEL
LIN {X 0,Y 457.23,Z 311.548,A -85,B 0,C 180,E1 -8760.513,E2 -8760.513} C_VEL
LIN {X 0,Y 455.703,Z 308.113,A -85,B 0,C 180,E1 -8760.729,E2 -8760.729} C_VEL
LIN {X 0,Y 451.447,Z 293.989,A -85,B 0,C 180,E1 -8762.791,E2 -8762.791} C_VEL
LIN {X 0,Y 447.204,Z 281.569,A -85,B 0,C 180,E1 -8764.74,E2 -8764.74} C_VEL
LIN {X 0,Y 446.439,Z 279.185,A -85,B 0,C 180,E1 -8765.138,E2 -8765.138} C_VEL
LIN {X 0,Y 446.429,Z 279.19,A -85,B 0,C 180,E1 -8768.082,E2 -8768.082} C_VEL
LIN {X 0,Y 446.427,Z 279.19,A -85,B 0,C 180,E1 -8770.918,E2 -8770.918} C_VEL
LIN {X 0,Y 446.422,Z 279.188,A -85,B 0,C 180,E1 -8773.844,E2 -8773.844} C_VEL
LIN {X 0,Y 446.399,Z 279.189,A -85,B 0,C 180,E1 -8776.404,E2 -8776.404} C_VEL
LIN {X 0,Y 446.426,Z 279.181,A -85,B 0,C 180,E1 -8779.083,E2 -8779.083} C_VEL
LIN {X 0,Y 446.415,Z 279.182,A -85,B 0,C 180,E1 -8781.921,E2 -8781.921} C_VEL
LIN {X 0,Y 446.429,Z 279.184,A -85,B 0,C 180,E1 -8785.477,E2 -8785.477} C_VEL
LIN {X 0,Y 446.416,Z 279.187,A -85,B 0,C 180,E1 -8788.7,E2 -8788.7} C_VEL
LIN {X 0,Y 446.485,Z 279.163,A -85,B 0,C 180,E1 -8791.822,E2 -8791.822} C_VEL
LIN {X 0,Y 446.459,Z 279.186,A -85,B 0,C 180,E1 -8794.848,E2 -8794.848} C_VEL
LIN {X 0,Y 446.449,Z 279.172,A -85,B 0,C 180,E1 -8798.246,E2 -8798.246} C_VEL
LIN {X 0,Y 446.458,Z 279.177,A -85,B 0,C 180,E1 -8801.65,E2 -8801.65} C_VEL
LIN {X 0,Y 446.509,Z 279.167,A -85,B 0,C 180,E1 -8804.48,E2 -8804.48} C_VEL
LIN {X 0,Y 446.518,Z 279.167,A -85,B 0,C 180,E1 -8808.194,E2 -8808.194} C_VEL
LIN {X 0,Y 446.533,Z 279.17,A -85,B 0,C 180,E1 -8810.945,E2 -8810.945} C_VEL
LIN {X 0,Y 446.615,Z 279.16,A -85,B 0,C 180,E1 -8813.676,E2 -8813.676} C_VEL
LIN {X 0,Y 446.684,Z 279.151,A -85,B 0,C 180,E1 -8817.295,E2 -8817.295} C_VEL
LIN {X 0,Y 446.789,Z 279.143,A -85,B 0,C 180,E1 -8820,E2 -8820} C_VEL
LIN {X 0,Y 446.657,Z 279.145,A -85,B 0,C 180,E1 -8822.706,E2 -8822.706} C_VEL
LIN {X 0,Y 446.613,Z 279.161,A -85,B 0,C 180,E1 -8826.325,E2 -8826.325} C_VEL
LIN {X 0,Y 446.528,Z 279.167,A -85,B 0,C 180,E1 -8829.056,E2 -8829.056} C_VEL
LIN {X 0,Y 446.524,Z 279.165,A -85,B 0,C 180,E1 -8832.73,E2 -8832.73} C_VEL
LIN {X 0,Y 446.457,Z 279.186,A -85,B 0,C 180,E1 -8836.209,E2 -8836.209} C_VEL
LIN {X 0,Y 446.471,Z 279.165,A -85,B 0,C 180,E1 -8839.304,E2 -8839.304} C_VEL
LIN {X 0,Y 446.413,Z 279.19,A -85,B 0,C 180,E1 -8842.2,E2 -8842.2} C_VEL
LIN {X 0,Y 446.415,Z 279.185,A -85,B 0,C 180,E1 -8845.155,E2 -8845.155} C_VEL
LIN {X 0,Y 446.417,Z 279.18,A -85,B 0,C 180,E1 -8848.184,E2 -8848.184} C_VEL
LIN {X 0,Y 446.391,Z 279.191,A -85,B 0,C 180,E1 -8851.303,E2 -8851.303} C_VEL
LIN {X 0,Y 446.413,Z 279.188,A -85,B 0,C 180,E1 -8854.525,E2 -8854.525} C_VEL
LIN {X 0,Y 446.388,Z 279.192,A -85,B 0,C 180,E1 -8857.882,E2 -8857.882} C_VEL
LIN {X 0,Y 446.397,Z 279.188,A -85,B 0,C 180,E1 -8860.913,E2 -8860.913} C_VEL
LIN {X 0,Y 446.462,Z 279.383,A -85,B 0,C 180,E1 -8864.512,E2 -8864.512} C_VEL
LIN {X 0,Y 448.94,Z 286.928,A -85,B 0,C 180,E1 -8865.782,E2 -8865.782} C_VEL
LIN {X 0,Y 458.488,Z 305.302,A -85,B 0,C 180,E1 -8866.924,E2 -8866.924} C_VEL
LIN {X 0,Y 462.376,Z 313.552,A -85,B 0,C 180,E1 -8867.383,E2 -8867.383} C_VEL
LIN {X 0,Y 459.067,Z 491.45,A -85,B 0,C 180,E1 -8870.342,E2 -8870.342} C_VEL
LIN {X 0,Y 458.39,Z 507.664,A -85,B 0,C 180,E1 -8870.769,E2 -8870.769} C_VEL
LIN {X 0,Y 457.536,Z 523.372,A -85,B 0,C 180,E1 -8871.354,E2 -8871.354} C_VEL
LIN {X 0,Y 456.464,Z 539.206,A -85,B 0,C 180,E1 -8872.125,E2 -8872.125} C_VEL
LIN {X 0,Y 455.237,Z 554.595,A -85,B 0,C 180,E1 -8873.07,E2 -8873.07} C_VEL
LIN {X 0,Y 454.489,Z 562.892,A -85,B 0,C 180,E1 -8873.67,E2 -8873.67} C_VEL
LIN {X 0,Y 453.417,Z 567.966,A -85,B 0,C 180,E1 -8874.03,E2 -8874.03} C_VEL
LIN {X 0,Y 449.943,Z 576.213,A -85,B 0,C 180,E1 -8874.577,E2 -8874.577} C_VEL
LIN {X 0,Y 446.442,Z 584.161,A -85,B 0,C 180,E1 -8875.186,E2 -8875.186} C_VEL
LIN {X 0,Y 445.341,Z 588.762,A -85,B 0,C 180,E1 -8875.638,E2 -8875.638} C_VEL
LIN {X 0,Y 443.973,Z 600.795,A -85,B 0,C 180,E1 -8877.034,E2 -8877.034} C_VEL
LIN {X 0,Y 442.674,Z 612.302,A -85,B 0,C 180,E1 -8878.616,E2 -8878.616} C_VEL
LIN {X 0,Y 441.605,Z 622.009,A -85,B 0,C 180,E1 -8880.176,E2 -8880.176} C_VEL
LIN {X 0,Y 440.621,Z 631.388,A -85,B 0,C 180,E1 -8881.931,E2 -8881.931} C_VEL
LIN {X 0,Y 439.807,Z 640.362,A -85,B 0,C 180,E1 -8883.938,E2 -8883.938} C_VEL
LIN {X 0,Y 439.145,Z 648.223,A -85,B 0,C 180,E1 -8886.102,E2 -8886.102} C_VEL
LIN {X 0,Y 438.699,Z 654.542,A -85,B 0,C 180,E1 -8888.307,E2 -8888.307} C_VEL
LIN {X 0,Y 438.411,Z 658.968,A -85,B 0,C 180,E1 -8890.327,E2 -8890.327} C_VEL
LIN {X 0,Y 438.212,Z 662.108,A -85,B 0,C 180,E1 -8892.259,E2 -8892.259} C_VEL
LIN {X 0,Y 438.166,Z 664.159,A -85,B 0,C 180,E1 -8894.235,E2 -8894.235} C_VEL
LIN {X 0,Y 438.144,Z 665.103,A -85,B 0,C 180,E1 -8896.078,E2 -8896.078} C_VEL
LIN {X 0,Y 438.275,Z 665.078,A -85,B 0,C 180,E1 -8898.01,E2 -8898.01} C_VEL
LIN {X 0,Y 438.214,Z 664.081,A -85,B 0,C 180,E1 -8899.839,E2 -8899.839} C_VEL
LIN {X 0,Y 438.254,Z 662.121,A -85,B 0,C 180,E1 -8901.702,E2 -8901.702} C_VEL
LIN {X 0,Y 438.443,Z 658.974,A -85,B 0,C 180,E1 -8903.635,E2 -8903.635} C_VEL
LIN {X 0,Y 438.56,Z 655.172,A -85,B 0,C 180,E1 -8905.404,E2 -8905.404} C_VEL
LIN {X 0,Y 438.86,Z 650.065,A -85,B 0,C 180,E1 -8907.246,E2 -8907.246} C_VEL
LIN {X 0,Y 439.343,Z 643.873,A -85,B 0,C 180,E1 -8909.083,E2 -8909.083} C_VEL
LIN {X 0,Y 439.919,Z 636.391,A -85,B 0,C 180,E1 -8910.915,E2 -8910.915} C_VEL
LIN {X 0,Y 440.752,Z 627.452,A -85,B 0,C 180,E1 -8912.742,E2 -8912.742} C_VEL
LIN {X 0,Y 441.894,Z 616.86,A -85,B 0,C 180,E1 -8914.561,E2 -8914.561} C_VEL
LIN {X 0,Y 442.989,Z 605.999,A -85,B 0,C 180,E1 -8916.147,E2 -8916.147} C_VEL
LIN {X 0,Y 444.201,Z 593.235,A -85,B 0,C 180,E1 -8917.729,E2 -8917.729} C_VEL
LIN {X 0,Y 445.722,Z 579.058,A -85,B 0,C 180,E1 -8919.186,E2 -8919.186} C_VEL
LIN {X 0,Y 447.024,Z 564.71,A -85,B 0,C 180,E1 -8920.416,E2 -8920.416} C_VEL
LIN {X 0,Y 448.261,Z 550.628,A -85,B 0,C 180,E1 -8921.416,E2 -8921.416} C_VEL
LIN {X 0,Y 449.392,Z 535.47,A -85,B 0,C 180,E1 -8922.303,E2 -8922.303} C_VEL
LIN {X 0,Y 450.199,Z 522.593,A -85,B 0,C 180,E1 -8922.911,E2 -8922.911} C_VEL
LIN {X 0,Y 451.04,Z 505.905,A -85,B 0,C 180,E1 -8923.516,E2 -8923.516} C_VEL
LIN {X 0,Y 451.722,Z 489.416,A -85,B 0,C 180,E1 -8923.926,E2 -8923.926} C_VEL
LIN {X 0,Y 454.708,Z 315.992,A -85,B 0,C 180,E1 -8926.783,E2 -8926.783} C_VEL
LIN {X 0,Y 454.323,Z 314.156,A -85,B 0,C 180,E1 -8926.841,E2 -8926.841} C_VEL
LIN {X 0,Y 441.342,Z 286.435,A -85,B 0,C 180,E1 -8928.247,E2 -8928.247} C_VEL
LIN {X 0,Y 439.429,Z 280.062,A -85,B 0,C 180,E1 -8929.27,E2 -8929.27} C_VEL
LIN {X 0,Y 439.366,Z 280.062,A -85,B 0,C 180,E1 -8932.575,E2 -8932.575} C_VEL
LIN {X 0,Y 439.357,Z 280.06,A -85,B 0,C 180,E1 -8935.588,E2 -8935.588} C_VEL
LIN {X 0,Y 439.384,Z 280.067,A -85,B 0,C 180,E1 -8938.676,E2 -8938.676} C_VEL
LIN {X 0,Y 439.346,Z 280.07,A -85,B 0,C 180,E1 -8942.024,E2 -8942.024} C_VEL
LIN {X 0,Y 439.383,Z 280.059,A -85,B 0,C 180,E1 -8945.337,E2 -8945.337} C_VEL
LIN {X 0,Y 439.349,Z 280.067,A -85,B 0,C 180,E1 -8948.598,E2 -8948.598} C_VEL
LIN {X 0,Y 439.359,Z 280.065,A -85,B 0,C 180,E1 -8951.251,E2 -8951.251} C_VEL
LIN {X 0,Y 439.374,Z 280.064,A -85,B 0,C 180,E1 -8954.733,E2 -8954.733} C_VEL
LIN {X 0,Y 439.346,Z 280.067,A -85,B 0,C 180,E1 -8957.789,E2 -8957.789} C_VEL
LIN {X 0,Y 439.361,Z 280.063,A -85,B 0,C 180,E1 -8960.219,E2 -8960.219} C_VEL
LIN {X 0,Y 439.366,Z 280.037,A -85,B 0,C 180,E1 -8963.711,E2 -8963.711} C_VEL
LIN {X 0,Y 439.371,Z 280.062,A -85,B 0,C 180,E1 -8967.053,E2 -8967.053} C_VEL
LIN {X 0,Y 439.371,Z 280.057,A -85,B 0,C 180,E1 -8970.273,E2 -8970.273} C_VEL
LIN {X 0,Y 439.379,Z 280.069,A -85,B 0,C 180,E1 -8973.603,E2 -8973.603} C_VEL
LIN {X 0,Y 439.367,Z 280.057,A -85,B 0,C 180,E1 -8976.428,E2 -8976.428} C_VEL
LIN {X 0,Y 439.39,Z 280.066,A -85,B 0,C 180,E1 -8979.397,E2 -8979.397} C_VEL
LIN {X 0,Y 439.405,Z 280.053,A -85,B 0,C 180,E1 -8982.308,E2 -8982.308} C_VEL
LIN {X 0,Y 439.446,Z 280.057,A -85,B 0,C 180,E1 -8985.173,E2 -8985.173} C_VEL
LIN {X 0,Y 439.484,Z 280.043,A -85,B 0,C 180,E1 -8988.001,E2 -8988.001} C_VEL
LIN {X 0,Y 439.505,Z 280.051,A -85,B 0,C 180,E1 -8991.725,E2 -8991.725} C_VEL
LIN {X 0,Y 439.618,Z 280.023,A -85,B 0,C 180,E1 -8994.495,E2 -8994.495} C_VEL
LIN {X 0,Y 439.632,Z 280.031,A -85,B 0,C 180,E1 -8998.167,E2 -8998.167} C_VEL
LIN {X 0,Y 439.761,Z 280.005,A -85,B 0,C 180,E1 -9000,E2 -9000} C_VEL
LIN {X 0,Y 439.64,Z 280.03,A -85,B 0,C 180,E1 -9002.748,E2 -9002.748} C_VEL
LIN {X 0,Y 439.593,Z 280.026,A -85,B 0,C 180,E1 -9006.425,E2 -9006.425} C_VEL
LIN {X 0,Y 439.5,Z 280.047,A -85,B 0,C 180,E1 -9009.201,E2 -9009.201} C_VEL
LIN {X 0,Y 439.466,Z 280.053,A -85,B 0,C 180,E1 -9012.937,E2 -9012.937} C_VEL
LIN {X 0,Y 439.446,Z 280.054,A -85,B 0,C 180,E1 -9016.348,E2 -9016.348} C_VEL
LIN {X 0,Y 439.401,Z 280.064,A -85,B 0,C 180,E1 -9019.626,E2 -9019.626} C_VEL
LIN {X 0,Y 439.365,Z 280.065,A -85,B 0,C 180,E1 -9022.575,E2 -9022.575} C_VEL
LIN {X 0,Y 439.405,Z 280.064,A -85,B 0,C 180,E1 -9025.584,E2 -9025.584} C_VEL
LIN {X 0,Y 439.416,Z 280.06,A -85,B 0,C 180,E1 -9028.673,E2 -9028.673} C_VEL
LIN {X 0,Y 439.369,Z 280.066,A -85,B 0,C 180,E1 -9032.03,E2 -9032.03} C_VEL
LIN {X 0,Y 439.395,Z 280.061,A -85,B 0,C 180,E1 -9035.34,E2 -9035.34} C_VEL
LIN {X 0,Y 439.387,Z 280.065,A -85,B 0,C 180,E1 -9038.594,E2 -9038.594} C_VEL
LIN {X 0,Y 439.388,Z 280.062,A -85,B 0,C 180,E1 -9041.257,E2 -9041.257} C_VEL
LIN {X 0,Y 439.405,Z 280.06,A -85,B 0,C 180,E1 -9044.728,E2 -9044.728} C_VEL
LIN {X 0,Y 439.396,Z 280.061,A -85,B 0,C 180,E1 -9047.796,E2 -9047.796} C_VEL
LIN {X 0,Y 439.435,Z 280.06,A -85,B 0,C 180,E1 -9050.228,E2 -9050.228} C_VEL
LIN {X 0,Y 439.371,Z 280.066,A -85,B 0,C 180,E1 -9053.713,E2 -9053.713} C_VEL
LIN {X 0,Y 439.401,Z 280.078,A -85,B 0,C 180,E1 -9055.264,E2 -9055.264} C_VEL
LIN {X 0,Y 446.02,Z 301.544,A -85,B 0,C 180,E1 -9058.307,E2 -9058.307} C_VEL
LIN {X 0,Y 448.079,Z 308.63,A -85,B 0,C 180,E1 -9059.263,E2 -9059.263} C_VEL
LIN {X 0,Y 450.194,Z 313.721,A -85,B 0,C 180,E1 -9059.498,E2 -9059.498} C_VEL
LIN {X 0,Y 454.503,Z 339.095,A -85,B 0,C 180,E1 -9060.233,E2 -9060.233} C_VEL
LIN {X 0,Y 451.493,Z 514.497,A -85,B 0,C 180,E1 -9063.122,E2 -9063.122} C_VEL
LIN {X 0,Y 450.783,Z 530.408,A -85,B 0,C 180,E1 -9063.526,E2 -9063.526} C_VEL
LIN {X 0,Y 449.868,Z 546.862,A -85,B 0,C 180,E1 -9064.123,E2 -9064.123} C_VEL
LIN {X 0,Y 448.794,Z 562.424,A -85,B 0,C 180,E1 -9064.864,E2 -9064.864} C_VEL
LIN {X 0,Y 447.538,Z 577.943,A -85,B 0,C 180,E1 -9065.803,E2 -9065.803} C_VEL
LIN {X 0,Y 446.243,Z 591.66,A -85,B 0,C 180,E1 -9066.813,E2 -9066.813} C_VEL
LIN {X 0,Y 444.974,Z 604.896,A -85,B 0,C 180,E1 -9067.969,E2 -9067.969} C_VEL
LIN {X 0,Y 443.739,Z 617.478,A -85,B 0,C 180,E1 -9069.262,E2 -9069.262} C_VEL
LIN {X 0,Y 442.509,Z 629.775,A -85,B 0,C 180,E1 -9070.758,E2 -9070.758} C_VEL
LIN {X 0,Y 441.344,Z 641.191,A -85,B 0,C 180,E1 -9072.389,E2 -9072.389} C_VEL
LIN {X 0,Y 440.494,Z 650.982,A -85,B 0,C 180,E1 -9074.025,E2 -9074.025} C_VEL
LIN {X 0,Y 439.642,Z 660.458,A -85,B 0,C 180,E1 -9075.89,E2 -9075.89} C_VEL
LIN {X 0,Y 439.146,Z 667.799,A -85,B 0,C 180,E1 -9077.626,E2 -9077.626} C_VEL
LIN {X 0,Y 438.763,Z 674.121,A -85,B 0,C 180,E1 -9079.385,E2 -9079.385} C_VEL
LIN {X 0,Y 438.485,Z 679.553,A -85,B 0,C 180,E1 -9081.242,E2 -9081.242} C_VEL
LIN {X 0,Y 438.391,Z 682.912,A -85,B 0,C 180,E1 -9082.632,E2 -9082.632} C_VEL
LIN {X 0,Y 438.306,Z 686.372,A -85,B 0,C 180,E1 -9084.479,E2 -9084.479} C_VEL
LIN {X 0,Y 438.254,Z 688.88,A -85,B 0,C 180,E1 -9086.322,E2 -9086.322} C_VEL
LIN {X 0,Y 438.268,Z 690.3,A -85,B 0,C 180,E1 -9088.162,E2 -9088.162} C_VEL
LIN {X 0,Y 438.248,Z 690.837,A -85,B 0,C 180,E1 -9090,E2 -9090} C_VEL
LIN {X 0,Y 438.285,Z 690.317,A -85,B 0,C 180,E1 -9091.838,E2 -9091.838} C_VEL
LIN {X 0,Y 438.254,Z 688.914,A -85,B 0,C 180,E1 -9093.678,E2 -9093.678} C_VEL
LIN {X 0,Y 438.306,Z 686.436,A -85,B 0,C 180,E1 -9095.521,E2 -9095.521} C_VEL
LIN {X 0,Y 438.389,Z 683.029,A -85,B 0,C 180,E1 -9097.369,E2 -9097.369} C_VEL
LIN {X 0,Y 438.574,Z 677.199,A -85,B 0,C 180,E1 -9099.687,E2 -9099.687} C_VEL
LIN {X 0,Y 439.108,Z 669.555,A -85,B 0,C 180,E1 -9102.009,E2 -9102.009} C_VEL
LIN {X 0,Y 439.692,Z 660.919,A -85,B 0,C 180,E1 -9104.108,E2 -9104.108} C_VEL
LIN {X 0,Y 440.588,Z 651.634,A -85,B 0,C 180,E1 -9105.972,E2 -9105.972} C_VEL
LIN {X 0,Y 441.457,Z 642.117,A -85,B 0,C 180,E1 -9107.607,E2 -9107.607} C_VEL
LIN {X 0,Y 442.673,Z 631.064,A -85,B 0,C 180,E1 -9109.234,E2 -9109.234} C_VEL
LIN {X 0,Y 444.007,Z 618.409,A -85,B 0,C 180,E1 -9110.813,E2 -9110.813} C_VEL
LIN {X 0,Y 445.331,Z 605.889,A -85,B 0,C 180,E1 -9112.135,E2 -9112.135} C_VEL
LIN {X 0,Y 446.804,Z 591.714,A -85,B 0,C 180,E1 -9113.401,E2 -9113.401} C_VEL
LIN {X 0,Y 448.201,Z 578.02,A -85,B 0,C 180,E1 -9114.427,E2 -9114.427} C_VEL
LIN {X 0,Y 449.62,Z 562.192,A -85,B 0,C 180,E1 -9115.396,E2 -9115.396} C_VEL
LIN {X 0,Y 450.875,Z 545.682,A -85,B 0,C 180,E1 -9116.188,E2 -9116.188} C_VEL
LIN {X 0,Y 451.828,Z 530.138,A -85,B 0,C 180,E1 -9116.751,E2 -9116.751} C_VEL
LIN {X 0,Y 452.577,Z 513.867,A -85,B 0,C 180,E1 -9117.168,E2 -9117.168} C_VEL
LIN {X 0,Y 456.021,Z 339.516,A -85,B 0,C 180,E1 -9120.095,E2 -9120.095} C_VEL
LIN {X 0,Y 451.905,Z 315.358,A -85,B 0,C 180,E1 -9120.878,E2 -9120.878} C_VEL
LIN {X 0,Y 448.472,Z 307.884,A -85,B 0,C 180,E1 -9121.336,E2 -9121.336} C_VEL
LIN {X 0,Y 443.731,Z 292.49,A -85,B 0,C 180,E1 -9123.666,E2 -9123.666} C_VEL
LIN {X 0,Y 439.378,Z 280.07,A -85,B 0,C 180,E1 -9125.733,E2 -9125.733} C_VEL
LIN {X 0,Y 439.389,Z 280.064,A -85,B 0,C 180,E1 -9128.595,E2 -9128.595} C_VEL
LIN {X 0,Y 439.389,Z 280.061,A -85,B 0,C 180,E1 -9131.257,E2 -9131.257} C_VEL
LIN {X 0,Y 439.405,Z 280.056,A -85,B 0,C 180,E1 -9134.729,E2 -9134.729} C_VEL
LIN {X 0,Y 439.396,Z 280.058,A -85,B 0,C 180,E1 -9137.796,E2 -9137.796} C_VEL
LIN {X 0,Y 439.43,Z 280.058,A -85,B 0,C 180,E1 -9140.228,E2 -9140.228} C_VEL
LIN {X 0,Y 439.373,Z 280.064,A -85,B 0,C 180,E1 -9143.713,E2 -9143.713} C_VEL
LIN {X 0,Y 439.372,Z 280.055,A -85,B 0,C 180,E1 -9147.054,E2 -9147.054} C_VEL
LIN {X 0,Y 439.383,Z 280.064,A -85,B 0,C 180,E1 -9150.275,E2 -9150.275} C_VEL
LIN {X 0,Y 439.429,Z 280.058,A -85,B 0,C 180,E1 -9153.397,E2 -9153.397} C_VEL
LIN {X 0,Y 439.388,Z 280.054,A -85,B 0,C 180,E1 -9156.43,E2 -9156.43} C_VEL
LIN {X 0,Y 439.39,Z 280.064,A -85,B 0,C 180,E1 -9159.398,E2 -9159.398} C_VEL
LIN {X 0,Y 439.431,Z 280.047,A -85,B 0,C 180,E1 -9162.31,E2 -9162.31} C_VEL
LIN {X 0,Y 439.448,Z 280.057,A -85,B 0,C 180,E1 -9165.174,E2 -9165.174} C_VEL
LIN {X 0,Y 439.485,Z 280.046,A -85,B 0,C 180,E1 -9168.002,E2 -9168.002} C_VEL
LIN {X 0,Y 439.505,Z 280.047,A -85,B 0,C 180,E1 -9171.726,E2 -9171.726} C_VEL
LIN {X 0,Y 439.606,Z 280.024,A -85,B 0,C 180,E1 -9174.496,E2 -9174.496} C_VEL
LIN {X 0,Y 439.635,Z 280.032,A -85,B 0,C 180,E1 -9178.168,E2 -9178.168} C_VEL
LIN {X 0,Y 439.758,Z 280.018,A -85,B 0,C 180,E1 -9180,E2 -9180} C_VEL
LIN {X 0,Y 439.609,Z 280.023,A -85,B 0,C 180,E1 -9182.75,E2 -9182.75} C_VEL
LIN {X 0,Y 439.565,Z 280.036,A -85,B 0,C 180,E1 -9186.427,E2 -9186.427} C_VEL
LIN {X 0,Y 439.492,Z 280.043,A -85,B 0,C 180,E1 -9189.202,E2 -9189.202} C_VEL
LIN {X 0,Y 439.468,Z 280.042,A -85,B 0,C 180,E1 -9192.938,E2 -9192.938} C_VEL
LIN {X 0,Y 439.405,Z 280.066,A -85,B 0,C 180,E1 -9196.329,E2 -9196.329} C_VEL
LIN {X 0,Y 439.404,Z 280.047,A -85,B 0,C 180,E1 -9199.627,E2 -9199.627} C_VEL
LIN {X 0,Y 439.357,Z 280.064,A -85,B 0,C 180,E1 -9202.576,E2 -9202.576} C_VEL
LIN {X 0,Y 439.356,Z 280.066,A -85,B 0,C 180,E1 -9205.589,E2 -9205.589} C_VEL
LIN {X 0,Y 439.379,Z 280.058,A -85,B 0,C 180,E1 -9208.677,E2 -9208.677} C_VEL
LIN {X 0,Y 439.345,Z 280.063,A -85,B 0,C 180,E1 -9212.025,E2 -9212.025} C_VEL
LIN {X 0,Y 439.383,Z 280.06,A -85,B 0,C 180,E1 -9215.338,E2 -9215.338} C_VEL
LIN {X 0,Y 439.351,Z 280.065,A -85,B 0,C 180,E1 -9218.599,E2 -9218.599} C_VEL
LIN {X 0,Y 439.36,Z 280.064,A -85,B 0,C 180,E1 -9221.252,E2 -9221.252} C_VEL
LIN {X 0,Y 439.375,Z 280.175,A -85,B 0,C 180,E1 -9223.929,E2 -9223.929} C_VEL
LIN {X 0,Y 441.781,Z 287.244,A -85,B 0,C 180,E1 -9225.153,E2 -9225.153} C_VEL
LIN {X 0,Y 451.552,Z 305.745,A -85,B 0,C 180,E1 -9226.362,E2 -9226.362} C_VEL
LIN {X 0,Y 456.345,Z 315.761,A -85,B 0,C 180,E1 -9226.944,E2 -9226.944} C_VEL
LIN {X 0,Y 452.836,Z 492.982,A -85,B 0,C 180,E1 -9229.935,E2 -9229.935} C_VEL
LIN {X 0,Y 452.046,Z 509.784,A -85,B 0,C 180,E1 -9230.399,E2 -9230.399} C_VEL
LIN {X 0,Y 451.165,Z 525.133,A -85,B 0,C 180,E1 -9231.001,E2 -9231.001} C_VEL
LIN {X 0,Y 449.976,Z 541.5,A -85,B 0,C 180,E1 -9231.836,E2 -9231.836} C_VEL
LIN {X 0,Y 448.788,Z 555.387,A -85,B 0,C 180,E1 -9232.713,E2 -9232.713} C_VEL
LIN {X 0,Y 447.274,Z 570.693,A -85,B 0,C 180,E1 -9233.897,E2 -9233.897} C_VEL
LIN {X 0,Y 445.812,Z 584.303,A -85,B 0,C 180,E1 -9235.17,E2 -9235.17} C_VEL
LIN {X 0,Y 445.341,Z 588.762,A -85,B 0,C 180,E1 -9235.638,E2 -9235.638} C_VEL
LIN {X 0,Y 444.245,Z 593.348,A -85,B 0,C 180,E1 -9236.106,E2 -9236.106} C_VEL
LIN {X 0,Y 440.652,Z 600.758,A -85,B 0,C 180,E1 -9236.842,E2 -9236.842} C_VEL
LIN {X 0,Y 437.092,Z 607.761,A -85,B 0,C 180,E1 -9237.624,E2 -9237.624} C_VEL
LIN {X 0,Y 436.011,Z 611.696,A -85,B 0,C 180,E1 -9238.168,E2 -9238.168} C_VEL
LIN {X 0,Y 434.76,Z 622.521,A -85,B 0,C 180,E1 -9239.926,E2 -9239.926} C_VEL
LIN {X 0,Y 433.708,Z 631.846,A -85,B 0,C 180,E1 -9241.707,E2 -9241.707} C_VEL
LIN {X 0,Y 432.895,Z 640.178,A -85,B 0,C 180,E1 -9243.6,E2 -9243.6} C_VEL
LIN {X 0,Y 432.22,Z 647.387,A -85,B 0,C 180,E1 -9245.586,E2 -9245.586} C_VEL
LIN {X 0,Y 431.737,Z 653.116,A -85,B 0,C 180,E1 -9247.509,E2 -9247.509} C_VEL
LIN {X 0,Y 431.436,Z 657.858,A -85,B 0,C 180,E1 -9249.498,E2 -9249.498} C_VEL
LIN {X 0,Y 431.267,Z 660.575,A -85,B 0,C 180,E1 -9250.978,E2 -9250.978} C_VEL
LIN {X 0,Y 431.107,Z 663.234,A -85,B 0,C 180,E1 -9252.936,E2 -9252.936} C_VEL
LIN {X 0,Y 431.055,Z 664.832,A -85,B 0,C 180,E1 -9254.878,E2 -9254.878} C_VEL
LIN {X 0,Y 431.082,Z 665.435,A -85,B 0,C 180,E1 -9256.806,E2 -9256.806} C_VEL
LIN {X 0,Y 431.153,Z 664.998,A -85,B 0,C 180,E1 -9258.72,E2 -9258.72} C_VEL
LIN {X 0,Y 431.097,Z 663.647,A -85,B 0,C 180,E1 -9260.617,E2 -9260.617} C_VEL
LIN {X 0,Y 431.235,Z 661.237,A -85,B 0,C 180,E1 -9262.508,E2 -9262.508} C_VEL
LIN {X 0,Y 431.45,Z 657.904,A -85,B 0,C 180,E1 -9264.391,E2 -9264.391} C_VEL
LIN {X 0,Y 431.764,Z 652.214,A -85,B 0,C 180,E1 -9266.734,E2 -9266.734} C_VEL
LIN {X 0,Y 432.259,Z 644.786,A -85,B 0,C 180,E1 -9269.068,E2 -9269.068} C_VEL
LIN {X 0,Y 432.941,Z 636.408,A -85,B 0,C 180,E1 -9271.163,E2 -9271.163} C_VEL
LIN {X 0,Y 433.7,Z 628.62,A -85,B 0,C 180,E1 -9272.786,E2 -9272.786} C_VEL
LIN {X 0,Y 434.701,Z 619.656,A -85,B 0,C 180,E1 -9274.404,E2 -9274.404} C_VEL
LIN {X 0,Y 435.852,Z 609.119,A -85,B 0,C 180,E1 -9276.016,E2 -9276.016} C_VEL
LIN {X 0,Y 437.153,Z 596.819,A -85,B 0,C 180,E1 -9277.622,E2 -9277.622} C_VEL
LIN {X 0,Y 438.488,Z 584.458,A -85,B 0,C 180,E1 -9278.99,E2 -9278.99} C_VEL
LIN {X 0,Y 439.777,Z 571.214,A -85,B 0,C 180,E1 -9280.241,E2 -9280.241} C_VEL
LIN {X 0,Y 441.19,Z 556.71,A -85,B 0,C 180,E1 -9281.369,E2 -9281.369} C_VEL
LIN {X 0,Y 442.334,Z 542.759,A -85,B 0,C 180,E1 -9282.269,E2 -9282.269} C_VEL
LIN {X 0,Y 443.344,Z 527.912,A -85,B 0,C 180,E1 -9283.055,E2 -9283.055} C_VEL
LIN {X 0,Y 444.373,Z 511.396,A -85,B 0,C 180,E1 -9283.723,E2 -9283.723} C_VEL
LIN {X 0,Y 445.1,Z 495.939,A -85,B 0,C 180,E1 -9284.166,E2 -9284.166} C_VEL
LIN {X 0,Y 445.618,Z 473.587,A -85,B 0,C 180,E1 -9284.587,E2 -9284.587} C_VEL
LIN {X 0,Y 448.432,Z 317.707,A -85,B 0,C 180,E1 -9287.173,E2 -9287.173} C_VEL
LIN {X 0,Y 447.409,Z 314.772,A -85,B 0,C 180,E1 -9287.296,E2 -9287.296} C_VEL
LIN {X 0,Y 434.128,Z 286.693,A -85,B 0,C 180,E1 -9288.763,E2 -9288.763} C_VEL
LIN {X 0,Y 432.355,Z 280.942,A -85,B 0,C 180,E1 -9289.7,E2 -9289.7} C_VEL
LIN {X 0,Y 432.315,Z 280.945,A -85,B 0,C 180,E1 -9292.964,E2 -9292.964} C_VEL
LIN {X 0,Y 432.309,Z 280.937,A -85,B 0,C 180,E1 -9296.036,E2 -9296.036} C_VEL
LIN {X 0,Y 432.324,Z 280.945,A -85,B 0,C 180,E1 -9299.189,E2 -9299.189} C_VEL
LIN {X 0,Y 432.308,Z 280.948,A -85,B 0,C 180,E1 -9302.444,E2 -9302.444} C_VEL
LIN {X 0,Y 432.331,Z 280.942,A -85,B 0,C 180,E1 -9305.818,E2 -9305.818} C_VEL
LIN {X 0,Y 432.3,Z 280.944,A -85,B 0,C 180,E1 -9309.348,E2 -9309.348} C_VEL
LIN {X 0,Y 432.302,Z 280.944,A -85,B 0,C 180,E1 -9311.801,E2 -9311.801} C_VEL
LIN {X 0,Y 432.333,Z 280.943,A -85,B 0,C 180,E1 -9314.347,E2 -9314.347} C_VEL
LIN {X 0,Y 432.302,Z 280.939,A -85,B 0,C 180,E1 -9317.018,E2 -9317.018} C_VEL
LIN {X 0,Y 432.289,Z 280.949,A -85,B 0,C 180,E1 -9319.828,E2 -9319.828} C_VEL
LIN {X 0,Y 432.296,Z 280.916,A -85,B 0,C 180,E1 -9323.02,E2 -9323.02} C_VEL
LIN {X 0,Y 432.334,Z 280.935,A -85,B 0,C 180,E1 -9326.002,E2 -9326.002} C_VEL
LIN {X 0,Y 432.343,Z 280.943,A -85,B 0,C 180,E1 -9329.491,E2 -9329.491} C_VEL
LIN {X 0,Y 432.321,Z 280.942,A -85,B 0,C 180,E1 -9331.872,E2 -9331.872} C_VEL
LIN {X 0,Y 432.323,Z 280.941,A -85,B 0,C 180,E1 -9334.996,E2 -9334.996} C_VEL
LIN {X 0,Y 432.36,Z 280.941,A -85,B 0,C 180,E1 -9338.045,E2 -9338.045} C_VEL
LIN {X 0,Y 432.385,Z 280.933,A -85,B 0,C 180,E1 -9341.029,E2 -9341.029} C_VEL
LIN {X 0,Y 432.431,Z 280.932,A -85,B 0,C 180,E1 -9343.961,E2 -9343.961} C_VEL
LIN {X 0,Y 432.46,Z 280.918,A -85,B 0,C 180,E1 -9347.803,E2 -9347.803} C_VEL
LIN {X 0,Y 432.465,Z 280.929,A -85,B 0,C 180,E1 -9351.589,E2 -9351.589} C_VEL
LIN {X 0,Y 432.594,Z 280.898,A -85,B 0,C 180,E1 -9354.406,E2 -9354.406} C_VEL
LIN {X 0,Y 432.601,Z 280.907,A -85,B 0,C 180,E1 -9358.138,E2 -9358.138} C_VEL
LIN {X 0,Y 432.731,Z 280.881,A -85,B 0,C 180,E1 -9359.999,E2 -9359.999} C_VEL
LIN {X 0,Y 432.592,Z 280.909,A -85,B 0,C 180,E1 -9362.793,E2 -9362.793} C_VEL
LIN {X 0,Y 432.587,Z 280.902,A -85,B 0,C 180,E1 -9365.594,E2 -9365.594} C_VEL
LIN {X 0,Y 432.483,Z 280.914,A -85,B 0,C 180,E1 -9368.409,E2 -9368.409} C_VEL
LIN {X 0,Y 432.459,Z 280.922,A -85,B 0,C 180,E1 -9372.196,E2 -9372.196} C_VEL
LIN {X 0,Y 432.43,Z 280.928,A -85,B 0,C 180,E1 -9376.038,E2 -9376.038} C_VEL
LIN {X 0,Y 432.386,Z 280.939,A -85,B 0,C 180,E1 -9379.485,E2 -9379.485} C_VEL
LIN {X 0,Y 432.319,Z 280.946,A -85,B 0,C 180,E1 -9382.964,E2 -9382.964} C_VEL
LIN {X 0,Y 432.364,Z 280.939,A -85,B 0,C 180,E1 -9386.032,E2 -9386.032} C_VEL
LIN {X 0,Y 432.342,Z 280.947,A -85,B 0,C 180,E1 -9389.187,E2 -9389.187} C_VEL
LIN {X 0,Y 432.322,Z 280.945,A -85,B 0,C 180,E1 -9392.443,E2 -9392.443} C_VEL
LIN {X 0,Y 432.344,Z 280.937,A -85,B 0,C 180,E1 -9395.632,E2 -9395.632} C_VEL
LIN {X 0,Y 432.349,Z 280.943,A -85,B 0,C 180,E1 -9398.716,E2 -9398.716} C_VEL
LIN {X 0,Y 432.334,Z 280.943,A -85,B 0,C 180,E1 -9401.796,E2 -9401.796} C_VEL
LIN {X 0,Y 432.34,Z 280.939,A -85,B 0,C 180,E1 -9404.346,E2 -9404.346} C_VEL
LIN {X 0,Y 432.323,Z 280.942,A -85,B 0,C 180,E1 -9407.015,E2 -9407.015} C_VEL
LIN {X 0,Y 432.34,Z 280.943,A -85,B 0,C 180,E1 -9409.819,E2 -9409.819} C_VEL
LIN {X 0,Y 432.304,Z 280.948,A -85,B 0,C 180,E1 -9413.022,E2 -9413.022} C_VEL
LIN {X 0,Y 432.395,Z 281.112,A -85,B 0,C 180,E1 -9414.841,E2 -9414.841} C_VEL
LIN {X 0,Y 438.272,Z 300.206,A -85,B 0,C 180,E1 -9417.61,E2 -9417.61} C_VEL
LIN {X 0,Y 440.807,Z 308.493,A -85,B 0,C 180,E1 -9418.755,E2 -9418.755} C_VEL
LIN {X 0,Y 444.187,Z 316.46,A -85,B 0,C 180,E1 -9419.136,E2 -9419.136} C_VEL
LIN {X 0,Y 448.144,Z 339.609,A -85,B 0,C 180,E1 -9419.822,E2 -9419.822} C_VEL
LIN {X 0,Y 445.114,Z 512.664,A -85,B 0,C 180,E1 -9422.709,E2 -9422.709} C_VEL
LIN {X 0,Y 444.385,Z 529.124,A -85,B 0,C 180,E1 -9423.114,E2 -9423.114} C_VEL
LIN {X 0,Y 443.512,Z 544.596,A -85,B 0,C 180,E1 -9423.66,E2 -9423.66} C_VEL
LIN {X 0,Y 442.298,Z 561.656,A -85,B 0,C 180,E1 -9424.468,E2 -9424.468} C_VEL
LIN {X 0,Y 440.962,Z 577.16,A -85,B 0,C 180,E1 -9425.412,E2 -9425.412} C_VEL
LIN {X 0,Y 439.606,Z 591.06,A -85,B 0,C 180,E1 -9426.442,E2 -9426.442} C_VEL
LIN {X 0,Y 438.159,Z 605.556,A -85,B 0,C 180,E1 -9427.732,E2 -9427.732} C_VEL
LIN {X 0,Y 436.877,Z 617.971,A -85,B 0,C 180,E1 -9429.037,E2 -9429.037} C_VEL
LIN {X 0,Y 435.502,Z 631.141,A -85,B 0,C 180,E1 -9430.681,E2 -9430.681} C_VEL
LIN {X 0,Y 434.324,Z 642.333,A -85,B 0,C 180,E1 -9432.341,E2 -9432.341} C_VEL
LIN {X 0,Y 433.427,Z 651.893,A -85,B 0,C 180,E1 -9433.999,E2 -9433.999} C_VEL
LIN {X 0,Y 432.566,Z 661.185,A -85,B 0,C 180,E1 -9435.895,E2 -9435.895} C_VEL
LIN {X 0,Y 432.039,Z 668.93,A -85,B 0,C 180,E1 -9437.791,E2 -9437.791} C_VEL
LIN {X 0,Y 431.581,Z 675.283,A -85,B 0,C 180,E1 -9439.681,E2 -9439.681} C_VEL
LIN {X 0,Y 431.379,Z 680.491,A -85,B 0,C 180,E1 -9441.569,E2 -9441.569} C_VEL
LIN {X 0,Y 431.317,Z 684.98,A -85,B 0,C 180,E1 -9443.691,E2 -9443.691} C_VEL
LIN {X 0,Y 431.207,Z 687.516,A -85,B 0,C 180,E1 -9445.326,E2 -9445.326} C_VEL
LIN {X 0,Y 431.215,Z 689.478,A -85,B 0,C 180,E1 -9447.198,E2 -9447.198} C_VEL
LIN {X 0,Y 431.164,Z 690.472,A -85,B 0,C 180,E1 -9449.066,E2 -9449.066} C_VEL
LIN {X 0,Y 431.166,Z 690.481,A -85,B 0,C 180,E1 -9450.934,E2 -9450.934} C_VEL
LIN {X 0,Y 431.214,Z 689.541,A -85,B 0,C 180,E1 -9452.803,E2 -9452.803} C_VEL
LIN {X 0,Y 431.207,Z 687.605,A -85,B 0,C 180,E1 -9454.674,E2 -9454.674} C_VEL
LIN {X 0,Y 431.289,Z 684.685,A -85,B 0,C 180,E1 -9456.55,E2 -9456.55} C_VEL
LIN {X 0,Y 431.365,Z 680.715,A -85,B 0,C 180,E1 -9458.432,E2 -9458.432} C_VEL
LIN {X 0,Y 431.582,Z 675.629,A -85,B 0,C 180,E1 -9460.319,E2 -9460.319} C_VEL
LIN {X 0,Y 432.085,Z 669.422,A -85,B 0,C 180,E1 -9462.207,E2 -9462.207} C_VEL
LIN {X 0,Y 432.69,Z 660.812,A -85,B 0,C 180,E1 -9464.342,E2 -9464.342} C_VEL
LIN {X 0,Y 433.677,Z 651.568,A -85,B 0,C 180,E1 -9466.233,E2 -9466.233} C_VEL
LIN {X 0,Y 434.726,Z 640.601,A -85,B 0,C 180,E1 -9468.132,E2 -9468.132} C_VEL
LIN {X 0,Y 436.092,Z 629.289,A -85,B 0,C 180,E1 -9469.782,E2 -9469.782} C_VEL
LIN {X 0,Y 437.465,Z 617.262,A -85,B 0,C 180,E1 -9471.286,E2 -9471.286} C_VEL
LIN {X 0,Y 439.019,Z 603.659,A -85,B 0,C 180,E1 -9472.719,E2 -9472.719} C_VEL
LIN {X 0,Y 440.444,Z 590.503,A -85,B 0,C 180,E1 -9473.885,E2 -9473.885} C_VEL
LIN {X 0,Y 442.068,Z 575.15,A -85,B 0,C 180,E1 -9475.017,E2 -9475.017} C_VEL
LIN {X 0,Y 443.422,Z 560.513,A -85,B 0,C 180,E1 -9475.903,E2 -9475.903} C_VEL
LIN {X 0,Y 444.685,Z 544.968,A -85,B 0,C 180,E1 -9476.644,E2 -9476.644} C_VEL
LIN {X 0,Y 445.654,Z 529.225,A -85,B 0,C 180,E1 -9477.215,E2 -9477.215} C_VEL
LIN {X 0,Y 446.441,Z 512.498,A -85,B 0,C 180,E1 -9477.637,E2 -9477.637} C_VEL
LIN {X 0,Y 450.04,Z 340.699,A -85,B 0,C 180,E1 -9480.557,E2 -9480.557} C_VEL
LIN {X 0,Y 446.22,Z 318.07,A -85,B 0,C 180,E1 -9481.308,E2 -9481.308} C_VEL
LIN {X 0,Y 441.272,Z 307.77,A -85,B 0,C 180,E1 -9481.952,E2 -9481.952} C_VEL
LIN {X 0,Y 436.156,Z 291.668,A -85,B 0,C 180,E1 -9484.483,E2 -9484.483} C_VEL
LIN {X 0,Y 432.325,Z 280.943,A -85,B 0,C 180,E1 -9486.342,E2 -9486.342} C_VEL
LIN {X 0,Y 432.355,Z 280.936,A -85,B 0,C 180,E1 -9489.342,E2 -9489.342} C_VEL
LIN {X 0,Y 432.334,Z 280.935,A -85,B 0,C 180,E1 -9491.797,E2 -9491.797} C_VEL
LIN {X 0,Y 432.34,Z 280.94,A -85,B 0,C 180,E1 -9494.347,E2 -9494.347} C_VEL
LIN {X 0,Y 432.32,Z 280.948,A -85,B 0,C 180,E1 -9497.016,E2 -9497.016} C_VEL
LIN {X 0,Y 432.336,Z 280.942,A -85,B 0,C 180,E1 -9499.821,E2 -9499.821} C_VEL
LIN {X 0,Y 432.306,Z 280.937,A -85,B 0,C 180,E1 -9503.023,E2 -9503.023} C_VEL
LIN {X 0,Y 432.359,Z 280.935,A -85,B 0,C 180,E1 -9505.997,E2 -9505.997} C_VEL
LIN {X 0,Y 432.348,Z 280.941,A -85,B 0,C 180,E1 -9509.49,E2 -9509.49} C_VEL
LIN {X 0,Y 432.392,Z 280.925,A -85,B 0,C 180,E1 -9512.929,E2 -9512.929} C_VEL
LIN {X 0,Y 432.372,Z 280.934,A -85,B 0,C 180,E1 -9516.024,E2 -9516.024} C_VEL
LIN {X 0,Y 432.352,Z 280.938,A -85,B 0,C 180,E1 -9519.047,E2 -9519.047} C_VEL
LIN {X 0,Y 432.378,Z 280.93,A -85,B 0,C 180,E1 -9522.012,E2 -9522.012} C_VEL
LIN {X 0,Y 432.396,Z 280.931,A -85,B 0,C 180,E1 -9524.927,E2 -9524.927} C_VEL
LIN {X 0,Y 432.46,Z 280.922,A -85,B 0,C 180,E1 -9527.804,E2 -9527.804} C_VEL
LIN {X 0,Y 432.465,Z 280.924,A -85,B 0,C 180,E1 -9531.59,E2 -9531.59} C_VEL
LIN {X 0,Y 432.58,Z 280.9,A -85,B 0,C 180,E1 -9534.406,E2 -9534.406} C_VEL
LIN {X 0,Y 432.604,Z 280.907,A -85,B 0,C 180,E1 -9538.139,E2 -9538.139} C_VEL
LIN {X 0,Y 432.728,Z 280.894,A -85,B 0,C 180,E1 -9540.001,E2 -9540.001} C_VEL
LIN {X 0,Y 432.562,Z 280.9,A -85,B 0,C 180,E1 -9542.794,E2 -9542.794} C_VEL
LIN {X 0,Y 432.579,Z 280.912,A -85,B 0,C 180,E1 -9545.595,E2 -9545.595} C_VEL
LIN {X 0,Y 432.464,Z 280.91,A -85,B 0,C 180,E1 -9548.411,E2 -9548.411} C_VEL
LIN {X 0,Y 432.462,Z 280.923,A -85,B 0,C 180,E1 -9552.197,E2 -9552.197} C_VEL
LIN {X 0,Y 432.392,Z 280.935,A -85,B 0,C 180,E1 -9556.041,E2 -9556.041} C_VEL
LIN {X 0,Y 432.389,Z 280.919,A -85,B 0,C 180,E1 -9559.485,E2 -9559.485} C_VEL
LIN {X 0,Y 432.305,Z 280.94,A -85,B 0,C 180,E1 -9562.966,E2 -9562.966} C_VEL
LIN {X 0,Y 432.308,Z 280.949,A -85,B 0,C 180,E1 -9566.037,E2 -9566.037} C_VEL
LIN {X 0,Y 432.317,Z 280.941,A -85,B 0,C 180,E1 -9569.19,E2 -9569.19} C_VEL
LIN {X 0,Y 432.307,Z 280.94,A -85,B 0,C 180,E1 -9572.445,E2 -9572.445} C_VEL
LIN {X 0,Y 432.332,Z 280.939,A -85,B 0,C 180,E1 -9575.819,E2 -9575.819} C_VEL
LIN {X 0,Y 432.301,Z 280.947,A -85,B 0,C 180,E1 -9579.349,E2 -9579.349} C_VEL
LIN {X 0,Y 432.303,Z 280.946,A -85,B 0,C 180,E1 -9581.801,E2 -9581.801} C_VEL
LIN {X 0,Y 432.315,Z 281.087,A -85,B 0,C 180,E1 -9583.342,E2 -9583.342} C_VEL
LIN {X 0,Y 434.485,Z 287.412,A -85,B 0,C 180,E1 -9584.478,E2 -9584.478} C_VEL
LIN {X 0,Y 444.835,Z 306.431,A -85,B 0,C 180,E1 -9585.799,E2 -9585.799} C_VEL
LIN {X 0,Y 450.408,Z 318.043,A -85,B 0,C 180,E1 -9586.498,E2 -9586.498} C_VEL
LIN {X 0,Y 446.68,Z 493.07,A -85,B 0,C 180,E1 -9589.487,E2 -9589.487} C_VEL
LIN {X 0,Y 445.857,Z 509.969,A -85,B 0,C 180,E1 -9589.96,E2 -9589.96} C_VEL
LIN {X 0,Y 444.99,Z 524.44,A -85,B 0,C 180,E1 -9590.529,E2 -9590.529} C_VEL
LIN {X 0,Y 443.851,Z 539.538,A -85,B 0,C 180,E1 -9591.285,E2 -9591.285} C_VEL
LIN {X 0,Y 442.577,Z 553.658,A -85,B 0,C 180,E1 -9592.168,E2 -9592.168} C_VEL
LIN {X 0,Y 441.043,Z 568.567,A -85,B 0,C 180,E1 -9593.304,E2 -9593.304} C_VEL
LIN {X 0,Y 439.585,Z 582.088,A -85,B 0,C 180,E1 -9594.547,E2 -9594.547} C_VEL
LIN {X 0,Y 438.155,Z 594.178,A -85,B 0,C 180,E1 -9595.847,E2 -9595.847} C_VEL
LIN {X 0,Y 436.671,Z 606.164,A -85,B 0,C 180,E1 -9597.373,E2 -9597.373} C_VEL
LIN {X 0,Y 436.011,Z 611.696,A -85,B 0,C 180,E1 -9598.168,E2 -9598.168} C_VEL
LIN {X 0,Y 434.955,Z 615.627,A -85,B 0,C 180,E1 -9598.733,E2 -9598.733} C_VEL
LIN {X 0,Y 431.472,Z 621.92,A -85,B 0,C 180,E1 -9599.636,E2 -9599.636} C_VEL
LIN {X 0,Y 427.981,Z 627.834,A -85,B 0,C 180,E1 -9600.592,E2 -9600.592} C_VEL
LIN {X 0,Y 426.931,Z 631.152,A -85,B 0,C 180,E1 -9601.233,E2 -9601.233} C_VEL
LIN {X 0,Y 425.99,Z 640.004,A -85,B 0,C 180,E1 -9603.251,E2 -9603.251} C_VEL
LIN {X 0,Y 425.329,Z 646.474,A -85,B 0,C 180,E1 -9605.023,E2 -9605.023} C_VEL
LIN {X 0,Y 424.738,Z 652.815,A -85,B 0,C 180,E1 -9607.117,E2 -9607.117} C_VEL
LIN {X 0,Y 424.426,Z 657.628,A -85,B 0,C 180,E1 -9609.144,E2 -9609.144} C_VEL
LIN {X 0,Y 424.209,Z 660.701,A -85,B 0,C 180,E1 -9610.795,E2 -9610.795} C_VEL
LIN {X 0,Y 424.027,Z 663.211,A -85,B 0,C 180,E1 -9612.642,E2 -9612.642} C_VEL
LIN {X 0,Y 423.975,Z 664.943,A -85,B 0,C 180,E1 -9614.62,E2 -9614.62} C_VEL
LIN {X 0,Y 423.971,Z 665.612,A -85,B 0,C 180,E1 -9616.581,E2 -9616.581} C_VEL
LIN {X 0,Y 424.081,Z 665.303,A -85,B 0,C 180,E1 -9618.529,E2 -9618.529} C_VEL
LIN {X 0,Y 423.997,Z 664.016,A -85,B 0,C 180,E1 -9620.459,E2 -9620.459} C_VEL
LIN {X 0,Y 424.123,Z 661.738,A -85,B 0,C 180,E1 -9622.382,E2 -9622.382} C_VEL
LIN {X 0,Y 424.357,Z 658.472,A -85,B 0,C 180,E1 -9624.297,E2 -9624.297} C_VEL
LIN {X 0,Y 424.601,Z 654.137,A -85,B 0,C 180,E1 -9626.204,E2 -9626.204} C_VEL
LIN {X 0,Y 424.871,Z 648.791,A -85,B 0,C 180,E1 -9628.104,E2 -9628.104} C_VEL
LIN {X 0,Y 425.516,Z 642.145,A -85,B 0,C 180,E1 -9630,E2 -9630} C_VEL
LIN {X 0,Y 426.144,Z 634.26,A -85,B 0,C 180,E1 -9631.89,E2 -9631.89} C_VEL
LIN {X 0,Y 427.209,Z 624.878,A -85,B 0,C 180,E1 -9633.773,E2 -9633.773} C_VEL
LIN {X 0,Y 428.546,Z 613.726,A -85,B 0,C 180,E1 -9635.647,E2 -9635.647} C_VEL
LIN {X 0,Y 429.836,Z 602.167,A -85,B 0,C 180,E1 -9637.28,E2 -9637.28} C_VEL
LIN {X 0,Y 431.136,Z 590.593,A -85,B 0,C 180,E1 -9638.672,E2 -9638.672} C_VEL
LIN {X 0,Y 432.487,Z 578.329,A -85,B 0,C 180,E1 -9639.942,E2 -9639.942} C_VEL
LIN {X 0,Y 433.919,Z 563.8,A -85,B 0,C 180,E1 -9641.207,E2 -9641.207} C_VEL
LIN {X 0,Y 435.424,Z 547.664,A -85,B 0,C 180,E1 -9642.349,E2 -9642.349} C_VEL
LIN {X 0,Y 436.567,Z 532.644,A -85,B 0,C 180,E1 -9643.203,E2 -9643.203} C_VEL
LIN {X 0,Y 437.687,Z 516.017,A -85,B 0,C 180,E1 -9643.937,E2 -9643.937} C_VEL
LIN {X 0,Y 438.43,Z 500.596,A -85,B 0,C 180,E1 -9644.446,E2 -9644.446} C_VEL
LIN {X 0,Y 439.018,Z 483.975,A -85,B 0,C 180,E1 -9644.811,E2 -9644.811} C_VEL
LIN {X 0,Y 442.134,Z 319.227,A -85,B 0,C 180,E1 -9647.579,E2 -9647.579} C_VEL
LIN {X 0,Y 429.341,Z 292.046,A -85,B 0,C 180,E1 -9649.007,E2 -9649.007} C_VEL
LIN {X 0,Y 426.866,Z 286.819,A -85,B 0,C 180,E1 -9649.316,E2 -9649.316} C_VEL
LIN {X 0,Y 425.297,Z 281.822,A -85,B 0,C 180,E1 -9650.15,E2 -9650.15} C_VEL
LIN {X 0,Y 425.275,Z 281.826,A -85,B 0,C 180,E1 -9653.367,E2 -9653.367} C_VEL
LIN {X 0,Y 425.264,Z 281.816,A -85,B 0,C 180,E1 -9656.501,E2 -9656.501} C_VEL
LIN {X 0,Y 425.281,Z 281.822,A -85,B 0,C 180,E1 -9659.72,E2 -9659.72} C_VEL
LIN {X 0,Y 425.263,Z 281.824,A -85,B 0,C 180,E1 -9663.05,E2 -9663.05} C_VEL
LIN {X 0,Y 425.276,Z 281.822,A -85,B 0,C 180,E1 -9665.926,E2 -9665.926} C_VEL
LIN {X 0,Y 425.256,Z 281.821,A -85,B 0,C 180,E1 -9669.035,E2 -9669.035} C_VEL
LIN {X 0,Y 425.256,Z 281.821,A -85,B 0,C 180,E1 -9672.655,E2 -9672.655} C_VEL
LIN {X 0,Y 425.285,Z 281.819,A -85,B 0,C 180,E1 -9675.283,E2 -9675.283} C_VEL
LIN {X 0,Y 425.247,Z 281.825,A -85,B 0,C 180,E1 -9678.617,E2 -9678.617} C_VEL
LIN {X 0,Y 425.275,Z 281.814,A -85,B 0,C 180,E1 -9681.098,E2 -9681.098} C_VEL
LIN {X 0,Y 425.293,Z 281.799,A -85,B 0,C 180,E1 -9684.663,E2 -9684.663} C_VEL
LIN {X 0,Y 425.262,Z 281.826,A -85,B 0,C 180,E1 -9688.072,E2 -9688.072} C_VEL
LIN {X 0,Y 425.298,Z 281.81,A -85,B 0,C 180,E1 -9691.365,E2 -9691.365} C_VEL
LIN {X 0,Y 425.26,Z 281.82,A -85,B 0,C 180,E1 -9694.552,E2 -9694.552} C_VEL
LIN {X 0,Y 425.294,Z 281.818,A -85,B 0,C 180,E1 -9697.729,E2 -9697.729} C_VEL
LIN {X 0,Y 425.363,Z 281.807,A -85,B 0,C 180,E1 -9700.703,E2 -9700.703} C_VEL
LIN {X 0,Y 425.389,Z 281.806,A -85,B 0,C 180,E1 -9703.688,E2 -9703.688} C_VEL
LIN {X 0,Y 425.413,Z 281.797,A -85,B 0,C 180,E1 -9707.598,E2 -9707.598} C_VEL
LIN {X 0,Y 425.409,Z 281.81,A -85,B 0,C 180,E1 -9711.449,E2 -9711.449} C_VEL
LIN {X 0,Y 425.549,Z 281.775,A -85,B 0,C 180,E1 -9714.313,E2 -9714.313} C_VEL
LIN {X 0,Y 425.57,Z 281.783,A -85,B 0,C 180,E1 -9718.107,E2 -9718.107} C_VEL
LIN {X 0,Y 425.7,Z 281.756,A -85,B 0,C 180,E1 -9719.999,E2 -9719.999} C_VEL
LIN {X 0,Y 425.545,Z 281.787,A -85,B 0,C 180,E1 -9722.839,E2 -9722.839} C_VEL
LIN {X 0,Y 425.542,Z 281.779,A -85,B 0,C 180,E1 -9725.686,E2 -9725.686} C_VEL
LIN {X 0,Y 425.437,Z 281.792,A -85,B 0,C 180,E1 -9728.55,E2 -9728.55} C_VEL
LIN {X 0,Y 425.412,Z 281.8,A -85,B 0,C 180,E1 -9732.401,E2 -9732.401} C_VEL
LIN {X 0,Y 425.387,Z 281.805,A -85,B 0,C 180,E1 -9736.311,E2 -9736.311} C_VEL
LIN {X 0,Y 425.328,Z 281.817,A -85,B 0,C 180,E1 -9739.635,E2 -9739.635} C_VEL
LIN {X 0,Y 425.307,Z 281.823,A -85,B 0,C 180,E1 -9743.365,E2 -9743.365} C_VEL
LIN {X 0,Y 425.346,Z 281.817,A -85,B 0,C 180,E1 -9746.844,E2 -9746.844} C_VEL
LIN {X 0,Y 425.29,Z 281.821,A -85,B 0,C 180,E1 -9749.719,E2 -9749.719} C_VEL
LIN {X 0,Y 425.281,Z 281.823,A -85,B 0,C 180,E1 -9753.048,E2 -9753.048} C_VEL
LIN {X 0,Y 425.283,Z 281.815,A -85,B 0,C 180,E1 -9755.929,E2 -9755.929} C_VEL
LIN {X 0,Y 425.299,Z 281.823,A -85,B 0,C 180,E1 -9759.044,E2 -9759.044} C_VEL
LIN {X 0,Y 425.277,Z 281.826,A -85,B 0,C 180,E1 -9762.652,E2 -9762.652} C_VEL
LIN {X 0,Y 425.267,Z 281.825,A -85,B 0,C 180,E1 -9766.045,E2 -9766.045} C_VEL
LIN {X 0,Y 425.283,Z 281.823,A -85,B 0,C 180,E1 -9769.479,E2 -9769.479} C_VEL
LIN {X 0,Y 425.276,Z 281.825,A -85,B 0,C 180,E1 -9772.488,E2 -9772.488} C_VEL
LIN {X 0,Y 425.322,Z 281.94,A -85,B 0,C 180,E1 -9774.371,E2 -9774.371} C_VEL
LIN {X 0,Y 430.833,Z 299.603,A -85,B 0,C 180,E1 -9777,E2 -9777} C_VEL
LIN {X 0,Y 433.478,Z 308.257,A -85,B 0,C 180,E1 -9778.225,E2 -9778.225} C_VEL
LIN {X 0,Y 438.187,Z 319.117,A -85,B 0,C 180,E1 -9778.765,E2 -9778.765} C_VEL
LIN {X 0,Y 441.896,Z 341.501,A -85,B 0,C 180,E1 -9779.432,E2 -9779.432} C_VEL
LIN {X 0,Y 438.616,Z 513.91,A -85,B 0,C 180,E1 -9782.344,E2 -9782.344} C_VEL
LIN {X 0,Y 437.851,Z 530.487,A -85,B 0,C 180,E1 -9782.777,E2 -9782.777} C_VEL
LIN {X 0,Y 436.799,Z 547.477,A -85,B 0,C 180,E1 -9783.417,E2 -9783.417} C_VEL
LIN {X 0,Y 435.618,Z 562.816,A -85,B 0,C 180,E1 -9784.177,E2 -9784.177} C_VEL
LIN {X 0,Y 434.289,Z 577.927,A -85,B 0,C 180,E1 -9785.118,E2 -9785.118} C_VEL
LIN {X 0,Y 432.718,Z 593.312,A -85,B 0,C 180,E1 -9786.298,E2 -9786.298} C_VEL
LIN {X 0,Y 431.343,Z 606.202,A -85,B 0,C 180,E1 -9787.487,E2 -9787.487} C_VEL
LIN {X 0,Y 429.933,Z 619.398,A -85,B 0,C 180,E1 -9788.923,E2 -9788.923} C_VEL
LIN {X 0,Y 428.676,Z 630.688,A -85,B 0,C 180,E1 -9790.361,E2 -9790.361} C_VEL
LIN {X 0,Y 427.389,Z 642.053,A -85,B 0,C 180,E1 -9792.067,E2 -9792.067} C_VEL
LIN {X 0,Y 426.484,Z 651.517,A -85,B 0,C 180,E1 -9793.731,E2 -9793.731} C_VEL
LIN {X 0,Y 425.559,Z 660.85,A -85,B 0,C 180,E1 -9795.657,E2 -9795.657} C_VEL
LIN {X 0,Y 425.012,Z 668.62,A -85,B 0,C 180,E1 -9797.586,E2 -9797.586} C_VEL
LIN {X 0,Y 424.541,Z 675.003,A -85,B 0,C 180,E1 -9799.508,E2 -9799.508} C_VEL
LIN {X 0,Y 424.287,Z 680.23,A -85,B 0,C 180,E1 -9801.427,E2 -9801.427} C_VEL
LIN {X 0,Y 424.222,Z 684.985,A -85,B 0,C 180,E1 -9803.72,E2 -9803.72} C_VEL
LIN {X 0,Y 424.133,Z 687.282,A -85,B 0,C 180,E1 -9805.248,E2 -9805.248} C_VEL
LIN {X 0,Y 424.112,Z 689.251,A -85,B 0,C 180,E1 -9807.151,E2 -9807.151} C_VEL
LIN {X 0,Y 424.083,Z 690.261,A -85,B 0,C 180,E1 -9809.051,E2 -9809.051} C_VEL
LIN {X 0,Y 424.086,Z 690.277,A -85,B 0,C 180,E1 -9810.95,E2 -9810.95} C_VEL
LIN {X 0,Y 424.11,Z 689.351,A -85,B 0,C 180,E1 -9812.85,E2 -9812.85} C_VEL
LIN {X 0,Y 424.112,Z 687.422,A -85,B 0,C 180,E1 -9814.753,E2 -9814.753} C_VEL
LIN {X 0,Y 424.209,Z 684.517,A -85,B 0,C 180,E1 -9816.66,E2 -9816.66} C_VEL
LIN {X 0,Y 424.276,Z 680.557,A -85,B 0,C 180,E1 -9818.574,E2 -9818.574} C_VEL
LIN {X 0,Y 424.548,Z 675.497,A -85,B 0,C 180,E1 -9820.492,E2 -9820.492} C_VEL
LIN {X 0,Y 425.062,Z 669.311,A -85,B 0,C 180,E1 -9822.412,E2 -9822.412} C_VEL
LIN {X 0,Y 425.722,Z 660.725,A -85,B 0,C 180,E1 -9824.581,E2 -9824.581} C_VEL
LIN {X 0,Y 426.766,Z 651.508,A -85,B 0,C 180,E1 -9826.504,E2 -9826.504} C_VEL
LIN {X 0,Y 427.878,Z 640.583,A -85,B 0,C 180,E1 -9828.433,E2 -9828.433} C_VEL
LIN {X 0,Y 429.322,Z 629.333,A -85,B 0,C 180,E1 -9830.107,E2 -9830.107} C_VEL
LIN {X 0,Y 430.805,Z 617.227,A -85,B 0,C 180,E1 -9831.649,E2 -9831.649} C_VEL
LIN {X 0,Y 432.435,Z 603.805,A -85,B 0,C 180,E1 -9833.084,E2 -9833.084} C_VEL
LIN {X 0,Y 433.956,Z 590.725,A -85,B 0,C 180,E1 -9834.265,E2 -9834.265} C_VEL
LIN {X 0,Y 435.574,Z 576.106,A -85,B 0,C 180,E1 -9835.371,E2 -9835.371} C_VEL
LIN {X 0,Y 437.086,Z 561.011,A -85,B 0,C 180,E1 -9836.307,E2 -9836.307} C_VEL
LIN {X 0,Y 438.521,Z 544.329,A -85,B 0,C 180,E1 -9837.114,E2 -9837.114} C_VEL
LIN {X 0,Y 439.516,Z 528.562,A -85,B 0,C 180,E1 -9837.688,E2 -9837.688} C_VEL
LIN {X 0,Y 440.369,Z 511.407,A -85,B 0,C 180,E1 -9838.116,E2 -9838.116} C_VEL
LIN {X 0,Y 444.028,Z 341.087,A -85,B 0,C 180,E1 -9841.055,E2 -9841.055} C_VEL
LIN {X 0,Y 440.532,Z 320.842,A -85,B 0,C 180,E1 -9841.753,E2 -9841.753} C_VEL
LIN {X 0,Y 434.004,Z 307.359,A -85,B 0,C 180,E1 -9842.643,E2 -9842.643} C_VEL
LIN {X 0,Y 429.349,Z 293.175,A -85,B 0,C 180,E1 -9844.954,E2 -9844.954} C_VEL
LIN {X 0,Y 425.279,Z 281.818,A -85,B 0,C 180,E1 -9846.95,E2 -9846.95} C_VEL
LIN {X 0,Y 425.294,Z 281.822,A -85,B 0,C 180,E1 -9850.127,E2 -9850.127} C_VEL
LIN {X 0,Y 425.264,Z 281.828,A -85,B 0,C 180,E1 -9853.352,E2 -9853.352} C_VEL
LIN {X 0,Y 425.257,Z 281.825,A -85,B 0,C 180,E1 -9856.649,E2 -9856.649} C_VEL
LIN {X 0,Y 425.29,Z 281.82,A -85,B 0,C 180,E1 -9859.874,E2 -9859.874} C_VEL
LIN {X 0,Y 425.278,Z 281.811,A -85,B 0,C 180,E1 -9862.489,E2 -9862.489} C_VEL
LIN {X 0,Y 425.307,Z 281.813,A -85,B 0,C 180,E1 -9865.818,E2 -9865.818} C_VEL
LIN {X 0,Y 425.291,Z 281.822,A -85,B 0,C 180,E1 -9869.239,E2 -9869.239} C_VEL
LIN {X 0,Y 425.349,Z 281.796,A -85,B 0,C 180,E1 -9872.443,E2 -9872.443} C_VEL
LIN {X 0,Y 425.352,Z 281.808,A -85,B 0,C 180,E1 -9875.603,E2 -9875.603} C_VEL
LIN {X 0,Y 425.294,Z 281.81,A -85,B 0,C 180,E1 -9878.682,E2 -9878.682} C_VEL
LIN {X 0,Y 425.334,Z 281.809,A -85,B 0,C 180,E1 -9881.703,E2 -9881.703} C_VEL
LIN {X 0,Y 425.349,Z 281.804,A -85,B 0,C 180,E1 -9884.671,E2 -9884.671} C_VEL
LIN {X 0,Y 425.413,Z 281.799,A -85,B 0,C 180,E1 -9887.599,E2 -9887.599} C_VEL
LIN {X 0,Y 425.409,Z 281.803,A -85,B 0,C 180,E1 -9891.45,E2 -9891.45} C_VEL
LIN {X 0,Y 425.534,Z 281.779,A -85,B 0,C 180,E1 -9894.313,E2 -9894.313} C_VEL
LIN {X 0,Y 425.573,Z 281.783,A -85,B 0,C 180,E1 -9898.108,E2 -9898.108} C_VEL
LIN {X 0,Y 425.697,Z 281.769,A -85,B 0,C 180,E1 -9900.001,E2 -9900.001} C_VEL
LIN {X 0,Y 425.518,Z 281.777,A -85,B 0,C 180,E1 -9902.841,E2 -9902.841} C_VEL
LIN {X 0,Y 425.533,Z 281.79,A -85,B 0,C 180,E1 -9905.688,E2 -9905.688} C_VEL
LIN {X 0,Y 425.409,Z 281.789,A -85,B 0,C 180,E1 -9908.551,E2 -9908.551} C_VEL
LIN {X 0,Y 425.415,Z 281.797,A -85,B 0,C 180,E1 -9912.402,E2 -9912.402} C_VEL
LIN {X 0,Y 425.321,Z 281.811,A -85,B 0,C 180,E1 -9915.331,E2 -9915.331} C_VEL
LIN {X 0,Y 425.316,Z 281.804,A -85,B 0,C 180,E1 -9918.299,E2 -9918.299} C_VEL
LIN {X 0,Y 425.294,Z 281.819,A -85,B 0,C 180,E1 -9921.319,E2 -9921.319} C_VEL
LIN {X 0,Y 425.295,Z 281.811,A -85,B 0,C 180,E1 -9924.649,E2 -9924.649} C_VEL
LIN {X 0,Y 425.239,Z 281.82,A -85,B 0,C 180,E1 -9927.566,E2 -9927.566} C_VEL
LIN {X 0,Y 425.287,Z 281.82,A -85,B 0,C 180,E1 -9930.76,E2 -9930.76} C_VEL
LIN {X 0,Y 425.29,Z 281.822,A -85,B 0,C 180,E1 -9934.283,E2 -9934.283} C_VEL
LIN {X 0,Y 425.27,Z 281.824,A -85,B 0,C 180,E1 -9937.696,E2 -9937.696} C_VEL
LIN {X 0,Y 425.242,Z 281.826,A -85,B 0,C 180,E1 -9940.514,E2 -9940.514} C_VEL
LIN {X 0,Y 425.255,Z 281.835,A -85,B 0,C 180,E1 -9942.695,E2 -9942.695} C_VEL
LIN {X 0,Y 427.272,Z 287.646,A -85,B 0,C 180,E1 -9943.779,E2 -9943.779} C_VEL
LIN {X 0,Y 436.762,Z 304.833,A -85,B 0,C 180,E1 -9945.04,E2 -9945.04} C_VEL
LIN {X 0,Y 444.302,Z 319.911,A -85,B 0,C 180,E1 -9946.012,E2 -9946.012} C_VEL
LIN {X 0,Y 442.064,Z 423.561,A -85,B 0,C 180,E1 -9947.802,E2 -9947.802} C_VEL
LIN {X 0,Y 440.546,Z 493.862,A -85,B 0,C 180,E1 -9949.038,E2 -9949.038} C_VEL
LIN {X 0,Y 439.636,Z 511.311,A -85,B 0,C 180,E1 -9949.539,E2 -9949.539} C_VEL
LIN {X 0,Y 438.698,Z 526.13,A -85,B 0,C 180,E1 -9950.148,E2 -9950.148} C_VEL
LIN {X 0,Y 437.435,Z 541.468,A -85,B 0,C 180,E1 -9950.948,E2 -9950.948} C_VEL
LIN {X 0,Y 436.155,Z 554.809,A -85,B 0,C 180,E1 -9951.804,E2 -9951.804} C_VEL
LIN {X 0,Y 434.539,Z 569.603,A -85,B 0,C 180,E1 -9952.962,E2 -9952.962} C_VEL
LIN {X 0,Y 432.973,Z 583.293,A -85,B 0,C 180,E1 -9954.253,E2 -9954.253} C_VEL
LIN {X 0,Y 431.385,Z 595.93,A -85,B 0,C 180,E1 -9955.66,E2 -9955.66} C_VEL
LIN {X 0,Y 429.944,Z 606.824,A -85,B 0,C 180,E1 -9957.077,E2 -9957.077} C_VEL
LIN {X 0,Y 428.677,Z 616.755,A -85,B 0,C 180,E1 -9958.586,E2 -9958.586} C_VEL
LIN {X 0,Y 427.434,Z 627.213,A -85,B 0,C 180,E1 -9960.444,E2 -9960.444} C_VEL
LIN {X 0,Y 426.931,Z 631.152,A -85,B 0,C 180,E1 -9961.233,E2 -9961.233} C_VEL
LIN {X 0,Y 425.913,Z 634.359,A -85,B 0,C 180,E1 -9961.889,E2 -9961.889} C_VEL
LIN {X 0,Y 419.801,Z 643.195,A -85,B 0,C 180,E1 -9963.822,E2 -9963.822} C_VEL
LIN {X 0,Y 418.521,Z 645.832,A -85,B 0,C 180,E1 -9964.526,E2 -9964.526} C_VEL
LIN {X 0,Y 418.36,Z 646.637,A -85,B 0,C 180,E1 -9964.771,E2 -9964.771} C_VEL
LIN {X 0,Y 417.769,Z 652.501,A -85,B 0,C 180,E1 -9966.713,E2 -9966.713} C_VEL
LIN {X 0,Y 417.399,Z 657.405,A -85,B 0,C 180,E1 -9968.776,E2 -9968.776} C_VEL
LIN {X 0,Y 417.135,Z 660.903,A -85,B 0,C 180,E1 -9970.65,E2 -9970.65} C_VEL
LIN {X 0,Y 416.966,Z 663.196,A -85,B 0,C 180,E1 -9972.338,E2 -9972.338} C_VEL
LIN {X 0,Y 416.914,Z 665.052,A -85,B 0,C 180,E1 -9974.353,E2 -9974.353} C_VEL
LIN {X 0,Y 416.871,Z 665.789,A -85,B 0,C 180,E1 -9976.348,E2 -9976.348} C_VEL
LIN {X 0,Y 416.991,Z 665.606,A -85,B 0,C 180,E1 -9978.331,E2 -9978.331} C_VEL
LIN {X 0,Y 416.9,Z 664.38,A -85,B 0,C 180,E1 -9980.295,E2 -9980.295} C_VEL
LIN {X 0,Y 417.036,Z 662.226,A -85,B 0,C 180,E1 -9982.252,E2 -9982.252} C_VEL
LIN {X 0,Y 417.267,Z 659.023,A -85,B 0,C 180,E1 -9984.2,E2 -9984.2} C_VEL
LIN {X 0,Y 417.503,Z 654.822,A -85,B 0,C 180,E1 -9986.139,E2 -9986.139} C_VEL
LIN {X 0,Y 417.784,Z 649.549,A -85,B 0,C 180,E1 -9988.072,E2 -9988.072} C_VEL
LIN {X 0,Y 418.467,Z 643.04,A -85,B 0,C 180,E1 -9990,E2 -9990} C_VEL
LIN {X 0,Y 419.198,Z 634.225,A -85,B 0,C 180,E1 -9992.162,E2 -9992.162} C_VEL
LIN {X 0,Y 420.352,Z 624.777,A -85,B 0,C 180,E1 -9994.075,E2 -9994.075} C_VEL
LIN {X 0,Y 421.743,Z 613.554,A -85,B 0,C 180,E1 -9995.978,E2 -9995.978} C_VEL
LIN {X 0,Y 423.098,Z 601.939,A -85,B 0,C 180,E1 -9997.636,E2 -9997.636} C_VEL
LIN {X 0,Y 424.492,Z 590.271,A -85,B 0,C 180,E1 -9999.049,E2 -9999.049} C_VEL
LIN {X 0,Y 426.001,Z 576.651,A -85,B 0,C 180,E1 -10000.456,E2 -10000.456} C_VEL
LIN {X 0,Y 427.406,Z 563.265,A -85,B 0,C 180,E1 -10001.621,E2 -10001.621} C_VEL
LIN {X 0,Y 428.817,Z 548.712,A -85,B 0,C 180,E1 -10002.662,E2 -10002.662} C_VEL
LIN {X 0,Y 430.011,Z 533.916,A -85,B 0,C 180,E1 -10003.528,E2 -10003.528} C_VEL
LIN {X 0,Y 431.008,Z 519.165,A -85,B 0,C 180,E1 -10004.218,E2 -10004.218} C_VEL
LIN {X 0,Y 431.952,Z 502.81,A -85,B 0,C 180,E1 -10004.788,E2 -10004.788} C_VEL
LIN {X 0,Y 432.575,Z 485.494,A -85,B 0,C 180,E1 -10005.188,E2 -10005.188} C_VEL
LIN {X 0,Y 435.803,Z 320.992,A -85,B 0,C 180,E1 -10007.992,E2 -10007.992} C_VEL
LIN {X 0,Y 421.415,Z 290.727,A -85,B 0,C 180,E1 -10009.639,E2 -10009.639} C_VEL
LIN {X 0,Y 419.554,Z 286.981,A -85,B 0,C 180,E1 -10009.887,E2 -10009.887} C_VEL
LIN {X 0,Y 418.239,Z 282.703,A -85,B 0,C 180,E1 -10010.61,E2 -10010.61} C_VEL
LIN {X 0,Y 418.261,Z 282.702,A -85,B 0,C 180,E1 -10013.783,E2 -10013.783} C_VEL
LIN {X 0,Y 418.204,Z 282.702,A -85,B 0,C 180,E1 -10017.04,E2 -10017.04} C_VEL
LIN {X 0,Y 418.24,Z 282.704,A -85,B 0,C 180,E1 -10020.272,E2 -10020.272} C_VEL
LIN {X 0,Y 418.229,Z 282.703,A -85,B 0,C 180,E1 -10023.679,E2 -10023.679} C_VEL
LIN {X 0,Y 418.232,Z 282.699,A -85,B 0,C 180,E1 -10027.225,E2 -10027.225} C_VEL
LIN {X 0,Y 418.207,Z 282.7,A -85,B 0,C 180,E1 -10030.866,E2 -10030.866} C_VEL
LIN {X 0,Y 418.203,Z 282.703,A -85,B 0,C 180,E1 -10033.727,E2 -10033.727} C_VEL
LIN {X 0,Y 418.199,Z 282.695,A -85,B 0,C 180,E1 -10036.447,E2 -10036.447} C_VEL
LIN {X 0,Y 418.207,Z 282.702,A -85,B 0,C 180,E1 -10039.133,E2 -10039.133} C_VEL
LIN {X 0,Y 418.234,Z 282.667,A -85,B 0,C 180,E1 -10042.774,E2 -10042.774} C_VEL
LIN {X 0,Y 418.233,Z 282.696,A -85,B 0,C 180,E1 -10046.321,E2 -10046.321} C_VEL
LIN {X 0,Y 418.24,Z 282.695,A -85,B 0,C 180,E1 -10049.727,E2 -10049.727} C_VEL
LIN {X 0,Y 418.211,Z 282.7,A -85,B 0,C 180,E1 -10053.016,E2 -10053.016} C_VEL
LIN {X 0,Y 418.258,Z 282.686,A -85,B 0,C 180,E1 -10056.216,E2 -10056.216} C_VEL
LIN {X 0,Y 418.252,Z 282.699,A -85,B 0,C 180,E1 -10059.337,E2 -10059.337} C_VEL
LIN {X 0,Y 418.281,Z 282.683,A -85,B 0,C 180,E1 -10062.395,E2 -10062.395} C_VEL
LIN {X 0,Y 418.302,Z 282.694,A -85,B 0,C 180,E1 -10065.402,E2 -10065.402} C_VEL
LIN {X 0,Y 418.315,Z 282.678,A -85,B 0,C 180,E1 -10068.368,E2 -10068.368} C_VEL
LIN {X 0,Y 418.466,Z 282.667,A -85,B 0,C 180,E1 -10072.278,E2 -10072.278} C_VEL
LIN {X 0,Y 418.507,Z 282.652,A -85,B 0,C 180,E1 -10074.217,E2 -10074.217} C_VEL
LIN {X 0,Y 418.54,Z 282.659,A -85,B 0,C 180,E1 -10078.075,E2 -10078.075} C_VEL
LIN {X 0,Y 418.669,Z 282.631,A -85,B 0,C 180,E1 -10079.999,E2 -10079.999} C_VEL
LIN {X 0,Y 418.501,Z 282.665,A -85,B 0,C 180,E1 -10082.887,E2 -10082.887} C_VEL
LIN {X 0,Y 418.5,Z 282.654,A -85,B 0,C 180,E1 -10085.782,E2 -10085.782} C_VEL
LIN {X 0,Y 418.397,Z 282.67,A -85,B 0,C 180,E1 -10088.695,E2 -10088.695} C_VEL
LIN {X 0,Y 418.316,Z 282.687,A -85,B 0,C 180,E1 -10091.631,E2 -10091.631} C_VEL
LIN {X 0,Y 418.302,Z 282.691,A -85,B 0,C 180,E1 -10094.596,E2 -10094.596} C_VEL
LIN {X 0,Y 418.279,Z 282.695,A -85,B 0,C 180,E1 -10097.604,E2 -10097.604} C_VEL
